// TwinCAT 3 PLC project PLC1
// ProgramVersion: 3.1.4023.0
// libraries:
//   Tc2_Standard, * (Beckhoff Automation GmbH)
//   Tc2_System, * (Beckhoff Automation GmbH)
//   Tc2_Utilities, * (Beckhoff Automation GmbH)
//   Tc3_Database, * (Beckhoff Automation GmbH)
//   Tc3_EventLogger, * (Beckhoff Automation GmbH)
//   Tc3_Module, * (Beckhoff Automation GmbH)
// project tree:
//   DUTs/ aE_Mode.TcDUT, aE_ProcessState.TcDUT, aE_State.TcDUT, aS_AnalogAlarm.TcDUT, aS_AutoControl.TcDUT, aS_DBField.TcDUT, aT_Furnace.TcDUT, aT_Heater.TcDUT, aT_Tank.TcDUT, aT_Turbine.TcDUT, AutoCtrlCmds.TcDUT, Components.TcDUT, InStream.TcDUT, MainInterface.TcDUT, OutStream.TcDUT, aS_PidParameter.TcDUT, Parameters.TcDUT
//   GVLs/ AlarmLimit.TcGVL, Interfacex.TcGVL, Streams.TcGVL
//   / PlcDBTask.TcTTO, PlcTask.TcTTO
//   POUs/ AlarmManagement.TcPOU, AutoControl.TcPOU, PnID.TcPOU, SaveDatabase.TcPOU, TanksSimulation.TcPOU, UpdateInterface.TcPOU
//   POUs/FB/ aFb_Motor.TcPOU, aFB_Valve.TcPOU
// real-time tasks:
//   TASK PlcTask: cycle T#100000us, priority 20, ADS port 350
//   TASK PlcDBTask: cycle T#1ms, priority 21, ADS port 351
//   TASK PlcTask1: cycle T#1ms, priority 22, ADS port 352
// I/O:
//   DEVICE Device 1 (EtherCAT), AmsNetId 5.57.208.6.2.1
//     Term 1 (EK1200) [EK1200-5000 EtherCAT Power supply (2A E-Bus)]
//       Term 2 (EL1004) [EL1004 4Ch. Dig. Input 24V, 3ms]
//       Term 3 (EL2004) [EL2004 4Ch. Dig. Output 24V, 0.5A]
//       Term 8 (EL3054) [EL3054 4Ch. Ana. Input 4-20mA]
//       Term 4 (EL9011) [EL9011 End Terminal]
//   DEVICE Device 5 (COM Port) (disabled)
// variable links:
//   PLC1/PLC1 Instance <-> Device 1 (EtherCAT)/Term 1 (EK1200)/Term 2 (EL1004)
//     PlcTask Inputs/AutoControl.bEmerNC <-> Channel 4/Input
//     PlcTask Inputs/AutoControl.bStart <-> Channel 3/Input
//     PlcTask Inputs/PnID.bHI <-> Channel 2/Input
//     PlcTask Inputs/PnID.bLO <-> Channel 1/Input
//   PLC1/PLC1 Instance <-> Device 1 (EtherCAT)/Term 1 (EK1200)/Term 3 (EL2004)
//     PlcTask Outputs/AutoControl.bErr <-> Channel 4/Output
//     PlcTask Outputs/AutoControl.bRun <-> Channel 3/Output
//     PlcTask Outputs/PnID.bMotor1 <-> Channel 1/Output
//     PlcTask Outputs/PnID.bMotor2 <-> Channel 2/Output
//   PLC1/PLC1 Instance <-> Device 1 (EtherCAT)/Term 1 (EK1200)/Term 8 (EL3054)
//     PlcTask Inputs/PnID.CircularPumpFlow <-> AI Standard Channel 1/Value

CONFIGURATION PLC1
    RESOURCE PLC ON TwinCAT3
        TASK PlcDBTask(INTERVAL := T#1ms, PRIORITY := 21);
        TASK PlcTask(INTERVAL := T#100000us, PRIORITY := 20);
        PROGRAM SaveDatabase WITH PlcDBTask : SaveDatabase;
        PROGRAM AutoControl WITH PlcTask : AutoControl;
        PROGRAM PnID WITH PlcTask : PnID;
        PROGRAM AlarmManagement WITH PlcTask : AlarmManagement;
        PROGRAM UpdateInterface WITH PlcTask : UpdateInterface;
    END_RESOURCE
END_CONFIGURATION

// ---- DUTs/aE_Mode.TcDUT
{attribute 'qualified_only'}
{attribute 'strict'}
TYPE aE_Mode :
(
	Manual := 1,
	Auto := 2,
	Service := 3
);
END_TYPE

// ---- DUTs/aE_ProcessState.TcDUT
{attribute 'qualified_only'}
{attribute 'strict'}
TYPE aE_ProcessState :
(
	Error := 0,
	Init := 1,
	Enable := 2,
	Start := 3,
	SteadyState := 4,
	Stop := 5,
	Disable := 6,
	Reset := 7
);
END_TYPE

// ---- DUTs/aE_State.TcDUT
{attribute 'qualified_only'}
{attribute 'strict'}
TYPE aE_State :
(
	Fault := 0,
	Auto := 1,
	ManRun := 2,
	ManStop := 3
);
END_TYPE

// ---- DUTs/aS_AnalogAlarm.TcDUT
TYPE aS_AnalogAlarm :
STRUCT
	HIHI: REAL;
	HI: REAL;
	LO: REAL;
	LOLO: REAL;
	Deadband: REAL;
END_STRUCT
END_TYPE

// ---- DUTs/aS_AutoControl.TcDUT
TYPE aS_AutoControl :
STRUCT
	Start: BOOL;
	Stop: BOOL;
	Setpoint: LREAL;
	ControlSignal: LREAL;
	Switch: BYTE;
END_STRUCT
END_TYPE

// ---- DUTs/aS_DBField.TcDUT
TYPE aS_DBField :
STRUCT
	Id: LINT;
	Sync: BOOL;
	Timestamp: DT;
	FurTemp: REAL;
	FurInper: REAL;
	LphTemp: REAL;
	LphPress: REAL;
	LphInpress: REAL;
	LphInflow: REAL;
	DeaTemp: REAL;
	DeaPress: REAL;
	HphTemp: REAL;
	HphPress: REAL;
	HphInpress: REAL;
	HphInflow: REAL;
	BoiTemp: REAL;
	BoiPress: REAL;
	ConTemp: REAL;
	ConInflow: REAL;
	TurHtemp: REAL;
	TurItemp: REAL;
	TurLtemp: REAL;
	TurHpress: REAL;
	TurIpress: REAL;
	TurLpress: REAL;
	TurSpeed: REAL;
	
	PconMode: BYTE;
	PconRun: BOOL;
	PconVal: REAL;
	PconTime: DINT;
	PconAtime: DINT;
	PconFault: BOOL;
	
	PsupMode: BYTE;
	PsupRun: BOOL;
	PsupVal: REAL;
	PsupTime: DINT;
	PsupAtime: DINT;
	PsupFault: BOOL;
	
	PcirMode: BYTE;
	PcirRun: BOOL;
	PcirVal: REAL;
	PcirTime: DINT;
	PcirAtime: DINT;
	PcirFault: BOOL;
	
	F1Mode: BYTE;
	F1Run: BOOL;
	F1Val: REAL;
	F1Time: DINT;
	F1Atime: DINT;
	F1Fault: BOOL;
	
	F2Mode: BYTE;
	F2Run: BOOL;
	F2Val: REAL;
	F2Time: DINT;
	F2Atime: DINT;
	F2Fault: BOOL;
	
	F3Mode: BYTE;
	F3Run: BOOL;
	F3Val: REAL;
	F3Time: DINT;
	F3Atime: DINT;
	F3Fault: BOOL;
	
	VlphMode: BYTE;
	VlphRun: BOOL;
	VlphVal: REAL;
	VlphTime: DINT;
	VlphAtime: DINT;
	VlphFault: BOOL;
	
	VdeaMode: BYTE;
	VdeaRun: BOOL;
	VdeaVal: REAL;
	VdeaTime: DINT;
	VdeaAtime: DINT;
	VdeaFault: BOOL;
	
	VhphMode: BYTE;
	VhphRun: BOOL;
	VhphVal: REAL;
	VhphTime: DINT;
	VhphAtime: DINT;
	VhphFault: BOOL;
	
	VturMode: BYTE;
	VturRun: BOOL;
	VturVal: REAL;
	VturTime: DINT;
	VturAtime: DINT;
	VturFault: BOOL;
	
	PintMode: BYTE;
	PintRun: BOOL;
	PintVal: REAL;
	PintTime: DINT;
	PintAtime: DINT;
	PintFault: BOOL;
END_STRUCT
END_TYPE

// ---- DUTs/aT_Furnace.TcDUT
TYPE aT_Furnace :
STRUCT
	InPercent: REAL;
	Temperature: REAL;
END_STRUCT
END_TYPE

// ---- DUTs/aT_Heater.TcDUT
TYPE aT_Heater :
STRUCT
	InPressure: REAL;
	InFlow: REAL;
	Temperature: REAL;
	Pressure: REAL;
END_STRUCT
END_TYPE

// ---- DUTs/aT_Tank.TcDUT
TYPE aT_Tank :
STRUCT
	HI: BOOL;
	LO: BOOL;
	Level: REAL;
END_STRUCT
END_TYPE

// ---- DUTs/aT_Turbine.TcDUT
TYPE aT_Turbine :
STRUCT
	Rotation: REAL;
	HighPressure: REAL;
	ImmediatePressure: REAL;
	OutPressure: REAL;
	HighTemperature: REAL;
	ImmediateTemperature: REAL;
	OutTemperature: REAL;
END_STRUCT
END_TYPE

// ---- DUTs/AutoCtrlCmds.TcDUT
TYPE AutoCtrlCmds :
STRUCT
	Start: BOOL;
	Stop: BOOL;
	Emergency: BOOL;
	Reset: BOOL;
	
	ProcessReady: BOOL;
	ProcessRun: BOOL;
	ProcessFault: BOOL;
END_STRUCT
END_TYPE

// ---- DUTs/Components.TcDUT
TYPE Components :
STRUCT
	ForceFan1: aFb_Motor;
	ForceFan2: aFb_Motor;
	ForceFan3: aFb_Motor;
	
	CondensePump: aFb_Motor;
	SupplyPump: aFb_Motor;
	CircularPump: aFb_Motor;
	InterPump: aFb_Motor;

	LPHValve: aFb_Valve;
	AirEjValve: aFb_Valve;
	HPHValve: aFb_Valve;
	TurbineValve: aFb_Valve;
	
	Furnace: aT_Furnace;
	LPHeater: aT_Heater;
	Deaerator: aT_Heater;
	HPHeater: aT_Heater;
	Boiler: aT_Heater;
	Turbine: aT_Turbine;
	Condenser: aT_Heater;
	
	InterTank: aT_Tank;
END_STRUCT
END_TYPE

// ---- DUTs/InStream.TcDUT
TYPE InStream :
STRUCT
	ForceFan1_Speed: REAL;
	ForceFan2_Speed: REAL;
	ForceFan3_Speed: REAL;
	Furnace_Temp: REAL;
	CondensePump_Press: REAL;
	CondensePump_Flow: REAL;
	CondensePump_Speed: REAL;
	LPHeater_Temp: REAL;
	LPHeater_Press: REAL;
	AirEjector_Temp: REAL;
	AirEjector_Press: REAL;
	SupplyPump_Press: REAL;
	SupplyPump_Flow: REAL;
	SupplyPump_Speed: REAL;
	HPHeater_Temp: REAL;
	HPHeater_Press: REAL;
	Boiler_Temp: REAL;
	Boiler_Press: REAL;
	Turbine_Rotation: REAL;
	Turbine_HighPress: REAL;
	Turbine_ImmediatePress: REAL;
	Turbine_OutPress: REAL;
	Turbine_HighTemp: REAL;
	Turbine_ImmediateTemp: REAL;
	Turbine_OutTemp: REAL;
	Condenser_Temp: REAL;

END_STRUCT
END_TYPE

// ---- DUTs/MainInterface.TcDUT
TYPE MainInterface :
STRUCT
	Components: Components;
END_STRUCT
END_TYPE

// ---- DUTs/OutStream.TcDUT
TYPE OutStream :
STRUCT
	ForceFan1_SetSpeed: REAL;
	ForceFan2_SetSpeed: REAL;
	ForceFan3_SetSpeed: REAL;
	CondensePump_SetSpeed: REAL;
	SupplyPump_SetSpeed: REAL;
	CircularPump_OutFlow: REAL;
	LPHeaterValve_SetPercent: REAL;
	AirEjectorValve_SetPercent: REAL;
	HPHeaterValve_SetPercent: REAL;
	TurbineValve_SetPercent: REAL;
END_STRUCT
END_TYPE

// ---- DUTs/aS_PidParameter.TcDUT
TYPE aS_PidParameter :
STRUCT
	Kp: LREAL;
	Ti: LREAL;
	Td: LREAL;
	Tn: LREAL;
END_STRUCT
END_TYPE

// ---- DUTs/Parameters.TcDUT
TYPE Parameters :
STRUCT
	PID_CondensePump_Press: aS_PidParameter := (Kp:= 91.7, Ti:= 6.368, Td:= 0.1396, Tn:= 0.078);//(Kp:= 91.7, Ti:= 6.368, Td:= 0.1396, Tn:= 0.078);//(Kp:= 200, Ti:= 33.333, Td:= 0, Tn:= 0.05);
	PID_SupplyPump_Press: aS_PidParameter := (Kp:= 40, Ti:= 10, Td:= 0.05, Tn:= 0.05);//(Kp:= 40, Ti:= 8, Td:= 0.125, Tn:= 0.05);
	//PID_Condenser_Temp: aS_PidParameter := (Kp:= -40, Ti:= 53.333, Td:= 2.5, Tn:= 0.05);
	PID_LPHeater_Temp: aS_PidParameter := (Kp:= 0.015, Ti:= 3, Td:= 0, Tn:= 0.05);//(Kp:= 0.02, Ti:= 6.667, Td:= 2, Tn:= 0.5);
	PID_AirEjector_Temp: aS_PidParameter := (Kp:= 0.025, Ti:= 50, Td:= 0, Tn:= 0.05);//(Kp:= 0.0085, Ti:= 4.048, Td:= 0, Tn:= 0.5);
	PID_HPHeater_Temp: aS_PidParameter := (Kp:= 0.01, Ti:= 20, Td:= 0, Tn:= 0.05);//(Kp:= 0.0103, Ti:= 4.12, Td:= 0, Tn:= 0.5);
	PID_Turbine_Speed: aS_PidParameter := (Kp:= 0.003, Ti:= 30, Td:= 0, Tn:= 0.05);//(Kp:= 0.001, Ti:= 10, Td:= 100, Tn:= 100);
	PID_Boiler_Temp: aS_PidParameter := (Kp:= 8, Ti:= 100, Td:= 0.0625, Tn:= 0.05);//(Kp:= 7, Ti:= 20, Td:= 1.4286, Tn:= 0.05);// //(Kp:= 7, Ti:= 100, Td:= 0, Tn:= 0.05);
	
	MaxSpeed_CondensePump: REAL := 1485;
	MaxSpeed_SupplyPump: REAL := 5645;
	MaxSpeed_CircularPump: REAL := 1500;
	MaxSpeed_InterPump: REAL := 1500;	
	MaxSpeed_ForceFan1: REAL := 1485;
	MaxSpeed_ForceFan2: REAL := 1485;
	MaxSpeed_ForceFan3: REAL := 1485;
	
	Condenser_Htemp: REAL := 50;
	Condenser_Ltemp: REAL := 30;
	
	SampleTime: REAL := 0.1;
END_STRUCT
END_TYPE

// ---- GVLs/AlarmLimit.TcGVL
{attribute 'qualified_only'}
VAR_GLOBAL
	alLPHeaterTemp: aS_AnalogAlarm := (HIHI:= 160, HI:= 150, LO:= 130, LOLO:= 120, Deadband:= 5);
	alLPHeaterPress: aS_AnalogAlarm := (HIHI:= 34, HI:= 31, LO:= 25, LOLO:= 22, Deadband:= 1);
	alDeaeratorTemp: aS_AnalogAlarm := (HIHI:= 220, HI:= 210, LO:= 190, LOLO:= 180, Deadband:= 5);
	alHPHeaterTemp: aS_AnalogAlarm := (HIHI:= 315, HI:= 305, LO:= 285, LOLO:= 275, Deadband:= 5);
	alHPHeaterPress: aS_AnalogAlarm := (HIHI:= 315, HI:= 305, LO:= 285, LOLO:= 275, Deadband:= 5);
	alBoilerTemp: aS_AnalogAlarm := (HIHI:= 590, HI:= 580, LO:= 550, LOLO:= 540, Deadband:= 5);
	alCondenserTemp: aS_AnalogAlarm := (HIHI:= 80, HI:= 70, LO:= 10, LOLO:= 5, Deadband:= 5);
	alTurbineTemp: aS_AnalogAlarm := (HIHI:= 170, HI:= 160, LO:= 140, LOLO:= 130, Deadband:= 5);
	alTurbinePress: aS_AnalogAlarm := (HIHI:= 0.2, HI:= 0.1, LO:= 0.02, LOLO:= 0.01, Deadband:= 0.005);
	alTurbineRotation: aS_AnalogAlarm := (HIHI:= 3020, HI:= 3010, LO:= 2990, LOLO:= 2980, Deadband:= 5);

END_VAR

// ---- GVLs/Interfacex.TcGVL
{attribute 'qualified_only'}
VAR_GLOBAL
	ScadaInterface: MainInterface;
	AutoCtrlCmds: AutoCtrlCmds;
	Parameters: Parameters;
END_VAR

// ---- GVLs/Streams.TcGVL
{attribute 'qualified_only'}
VAR_GLOBAL
	OutStream AT %MD0: OutStream;
	InStream AT %MD10: InStream;
END_VAR

// ---- POUs/SaveDatabase.TcPOU
PROGRAM SaveDatabase
VAR
	fbPLCDBWrite : FB_PLCDBWriteEvt (sNetID := '', tTimeout := T#5S);
	myDBID : UDINT:=1;
	sMyTableName : T_MaxString:='Data';
	ColumnNames : ARRAY [0..91] OF STRING(50);
	insertData : aS_DBField;
	tcMessage : I_TcMessage;
	
	//Các biến tạo timestamp
	systime: GETSYSTEMTIME;
	currentTime: T_FILETIME;
	timestring: string;
	
	bFirstScan: BOOL;
	bExecute: BOOL;
	fbTon: TON;
	iID: LINT;
END_VAR

IF NOT bFirstScan THEN
	bFirstScan := TRUE;
	InitColumnNames();
END_IF

fbTon(IN:= NOT fbTon.Q, PT:= T#1S);	
IF fbTon.Q THEN
	UpdateData();
	bExecute := TRUE;
END_IF

IF bExecute AND bFirstScan THEN
	//UpdateData();
	IF fbPLCDBWrite.WriteStruct(
		hDBID:= myDBID,
		sTableName:= sMyTableName,
		pRecord:= ADR(insertData),
		cbRecord:= SIZEOF(insertData),
		pColumnNames:= ADR(ColumnNames) ,
		cbColumnNames:= SIZEOF(ColumnNames)
	)
	THEN
		IF fbPLCDBWrite.bError THEN
			tcMessage := fbPLCDBWrite.ipTcResult;
		ELSE
			iId := iId + 1;
			bExecute:= FALSE;
		END_IF
	END_IF	
	
END_IF

ACTION InitColumnNames:
ColumnNames[0] := 'Id';
ColumnNames[1] := 'Sync';
ColumnNames[2] := 'Timestamp';

ColumnNames[3] := 'FurTemp';
ColumnNames[4] := 'FurInper';
ColumnNames[5] := 'LphTemp';
ColumnNames[6] := 'LphPress';
ColumnNames[7] := 'LphInpress';
ColumnNames[8] := 'LphInflow';
ColumnNames[9] := 'DeaTemp';
ColumnNames[10] := 'DeaPress';
ColumnNames[11] := 'HphTemp';
ColumnNames[12] := 'HphPress';
ColumnNames[13] := 'HphInpress';
ColumnNames[14] := 'HphInflow';
ColumnNames[15] := 'BoiTemp';
ColumnNames[16] := 'BoiPress';
ColumnNames[17] := 'ConTemp';
ColumnNames[18] := 'ConInflow';
ColumnNames[19] := 'TurHtemp';
ColumnNames[20] := 'TurItemp';
ColumnNames[21] := 'TurLtemp';
ColumnNames[22] := 'TurHpress';
ColumnNames[23] := 'TurIpress';
ColumnNames[24] := 'TurLpress';
ColumnNames[25] := 'TurSpeed';

ColumnNames[26] := 'PconMode';
ColumnNames[27] := 'PconRun';
ColumnNames[28] := 'PconVal';
ColumnNames[29] := 'PconTime';
ColumnNames[30] := 'PconAtime';
ColumnNames[31] := 'PconFault';

ColumnNames[32] := 'PsupMode';
ColumnNames[33] := 'PsupRun';
ColumnNames[34] := 'PsupVal';
ColumnNames[35] := 'PsupTime';
ColumnNames[36] := 'PsupAtime';
ColumnNames[37] := 'PsupFault';

ColumnNames[38] := 'PcirMode';
ColumnNames[39] := 'PcirRun';
ColumnNames[40] := 'PcirVal';
ColumnNames[41] := 'PcirTime';
ColumnNames[42] := 'PcirAtime';
ColumnNames[43] := 'PcirFault';

ColumnNames[44] := 'F1Mode';
ColumnNames[45] := 'F1Run';
ColumnNames[46] := 'F1Val';
ColumnNames[47] := 'F1Time';
ColumnNames[48] := 'F1Atime';
ColumnNames[49] := 'F1Fault';

ColumnNames[50] := 'F2Mode';
ColumnNames[51] := 'F2Run';
ColumnNames[52] := 'F2Val';
ColumnNames[53] := 'F2Time';
ColumnNames[54] := 'F2Atime';
ColumnNames[55] := 'F2Fault';

ColumnNames[56] := 'F3Mode';
ColumnNames[57] := 'F3Run';
ColumnNames[58] := 'F3Val';
ColumnNames[59] := 'F3Time';
ColumnNames[60] := 'F3Atime';
ColumnNames[61] := 'F3Fault';

ColumnNames[62] := 'VlphMode';
ColumnNames[63] := 'VlphRun';
ColumnNames[64] := 'VlphVal';
ColumnNames[65] := 'VlphTime';
ColumnNames[66] := 'VlphAtime';
ColumnNames[67] := 'VlphFault';

ColumnNames[68] := 'VdeaMode';
ColumnNames[69] := 'VdeaRun';
ColumnNames[70] := 'VdeaVal';
ColumnNames[71] := 'VdeaTime';
ColumnNames[72] := 'VdeaAtime';
ColumnNames[73] := 'VdeaFault';

ColumnNames[74] := 'VhphMode';
ColumnNames[75] := 'VhphRun';
ColumnNames[76] := 'VhphVal';
ColumnNames[77] := 'VhphTime';
ColumnNames[78] := 'VhphAtime';
ColumnNames[79] := 'VhphFault';

ColumnNames[80] := 'VturMode';
ColumnNames[81] := 'VturRun';
ColumnNames[82] := 'VturVal';
ColumnNames[83] := 'VturTime';
ColumnNames[84] := 'VturAtime';
ColumnNames[85] := 'VturFault';

ColumnNames[86] := 'PintMode';
ColumnNames[87] := 'PintRun';
ColumnNames[88] := 'PintVal';
ColumnNames[89] := 'PintTime';
ColumnNames[90] := 'PintAtime';
ColumnNames[91] := 'PintFault';
END_ACTION

ACTION UpdateData:
systime(timeLoDW => currentTime.dwLowDateTime, timeHiDW => currentTime.dwHighDateTime);	
timestring:= DT_TO_STRING(FILETIME_TO_DT(currentTime));
timestring:= delete(timestring, 3, 1);
timestring:= replace(timestring, ' ', 1, 11);

insertData.Id := iID;
insertData.Sync := FALSE;
insertData.Timestamp:= FILETIME_TO_DT(currentTime);
insertData.FurTemp:= Interfacex.ScadaInterface.Components.Furnace.Temperature;
insertData.FurInper:= Interfacex.ScadaInterface.Components.Furnace.InPercent;
insertData.LphTemp:= Interfacex.ScadaInterface.Components.LPHeater.Temperature;
insertData.LphPress:= Interfacex.ScadaInterface.Components.LPHeater.Pressure;
insertData.LphInpress:= Interfacex.ScadaInterface.Components.LPHeater.InPressure;
insertData.LphInflow:= Interfacex.ScadaInterface.Components.LPHeater.InFlow;
insertData.DeaTemp:= Interfacex.ScadaInterface.Components.Deaerator.Temperature;
insertData.DeaPress:= Interfacex.ScadaInterface.Components.Deaerator.Pressure;
insertData.HphTemp:= Interfacex.ScadaInterface.Components.HPHeater.Temperature;
insertData.HphPress:= Interfacex.ScadaInterface.Components.HPHeater.Pressure;
insertData.HphInpress:= Interfacex.ScadaInterface.Components.HPHeater.InPressure;
insertData.HphInflow:= Interfacex.ScadaInterface.Components.HPHeater.InFlow;
insertData.BoiTemp:= Interfacex.ScadaInterface.Components.Boiler.Temperature;
insertData.BoiPress:= Interfacex.ScadaInterface.Components.Boiler.Pressure;
insertData.ConTemp:= Interfacex.ScadaInterface.Components.Condenser.Temperature;
insertData.ConInflow:= Interfacex.ScadaInterface.Components.Condenser.InFlow;
insertData.TurHtemp:= Interfacex.ScadaInterface.Components.Turbine.HighTemperature;
insertData.TurItemp:= Interfacex.ScadaInterface.Components.Turbine.ImmediateTemperature;
insertData.TurLtemp:= Interfacex.ScadaInterface.Components.Turbine.OutTemperature;
insertData.TurHpress:= Interfacex.ScadaInterface.Components.Turbine.HighPressure;
insertData.TurIpress:= Interfacex.ScadaInterface.Components.Turbine.ImmediatePressure;
insertData.TurLpress:= Interfacex.ScadaInterface.Components.Turbine.OutPressure;
insertData.TurSpeed:= Interfacex.ScadaInterface.Components.Turbine.Rotation;

insertData.PconMode:= INT_TO_BYTE(Interfacex.ScadaInterface.Components.CondensePump.Mode); 
insertData.PconRun:= Interfacex.ScadaInterface.Components.CondensePump.RunFeedback;
insertData.PconVal:= Interfacex.ScadaInterface.Components.CondensePump.ActualSpeed;
insertData.PconTime:= Interfacex.ScadaInterface.Components.CondensePump.Runtime;
insertData.PconAtime:= Interfacex.ScadaInterface.Components.CondensePump.AccRuntime;
insertData.PconFault:= Interfacex.ScadaInterface.Components.CondensePump.Fault;

insertData.PsupMode:= INT_TO_BYTE(Interfacex.ScadaInterface.Components.SupplyPump.Mode); 
insertData.PsupRun:= Interfacex.ScadaInterface.Components.SupplyPump.RunFeedback;
insertData.PsupVal:= Interfacex.ScadaInterface.Components.SupplyPump.ActualSpeed;
insertData.PsupTime:= Interfacex.ScadaInterface.Components.SupplyPump.Runtime;
insertData.PsupAtime:= Interfacex.ScadaInterface.Components.SupplyPump.AccRuntime;
insertData.PsupFault:= Interfacex.ScadaInterface.Components.SupplyPump.Fault;

insertData.PcirMode:= INT_TO_BYTE(Interfacex.ScadaInterface.Components.CircularPump.Mode); 
insertData.PcirRun:= Interfacex.ScadaInterface.Components.CircularPump.RunFeedback;
insertData.PcirVal:= Interfacex.ScadaInterface.Components.CircularPump.ActualSpeed;
insertData.PcirTime:= Interfacex.ScadaInterface.Components.CircularPump.Runtime;
insertData.PcirAtime:= Interfacex.ScadaInterface.Components.CircularPump.AccRuntime;
insertData.PcirFault:= Interfacex.ScadaInterface.Components.CircularPump.Fault;

insertData.F1Mode:= INT_TO_BYTE(Interfacex.ScadaInterface.Components.ForceFan1.Mode); 
insertData.F1Run:= Interfacex.ScadaInterface.Components.ForceFan1.RunFeedback;
insertData.F1Val:= Interfacex.ScadaInterface.Components.ForceFan1.ActualSpeed;
insertData.F1Time:= Interfacex.ScadaInterface.Components.ForceFan1.Runtime;
insertData.F1Atime:= Interfacex.ScadaInterface.Components.ForceFan1.AccRuntime;
insertData.F1Fault:= Interfacex.ScadaInterface.Components.ForceFan1.Fault;

insertData.F2Mode:= INT_TO_BYTE(Interfacex.ScadaInterface.Components.ForceFan2.Mode); 
insertData.F2Run:= Interfacex.ScadaInterface.Components.ForceFan2.RunFeedback;
insertData.F2Val:= Interfacex.ScadaInterface.Components.ForceFan2.ActualSpeed;
insertData.F2Time:= Interfacex.ScadaInterface.Components.ForceFan2.Runtime;
insertData.F2Atime:= Interfacex.ScadaInterface.Components.ForceFan2.AccRuntime;
insertData.F2Fault:= Interfacex.ScadaInterface.Components.ForceFan2.Fault;

insertData.F3Mode:= INT_TO_BYTE(Interfacex.ScadaInterface.Components.ForceFan3.Mode); 
insertData.F3Run:= Interfacex.ScadaInterface.Components.ForceFan3.RunFeedback;
insertData.F3Val:= Interfacex.ScadaInterface.Components.ForceFan3.ActualSpeed;
insertData.F3Time:= Interfacex.ScadaInterface.Components.ForceFan3.Runtime;
insertData.F3Atime:= Interfacex.ScadaInterface.Components.ForceFan3.AccRuntime;
insertData.F3Fault:= Interfacex.ScadaInterface.Components.ForceFan3.Fault;

insertData.VlphMode:= INT_TO_BYTE(Interfacex.ScadaInterface.Components.LPHValve.Mode); 
insertData.VlphRun:= Interfacex.ScadaInterface.Components.LPHValve.RunFeedback;
insertData.VlphVal:= Interfacex.ScadaInterface.Components.LPHValve.OpenPercent;
insertData.VlphTime:= Interfacex.ScadaInterface.Components.LPHValve.Runtime;
insertData.VlphAtime:= Interfacex.ScadaInterface.Components.LPHValve.AccRuntime;
insertData.VlphFault:= Interfacex.ScadaInterface.Components.LPHValve.Fault;

insertData.VdeaMode:= INT_TO_BYTE(Interfacex.ScadaInterface.Components.AirEjValve.Mode); 
insertData.VdeaRun:= Interfacex.ScadaInterface.Components.AirEjValve.RunFeedback;
insertData.VdeaVal:= Interfacex.ScadaInterface.Components.AirEjValve.OpenPercent;
insertData.VdeaTime:= Interfacex.ScadaInterface.Components.AirEjValve.Runtime;
insertData.VdeaAtime:= Interfacex.ScadaInterface.Components.AirEjValve.AccRuntime;
insertData.VdeaFault:= Interfacex.ScadaInterface.Components.AirEjValve.Fault;

insertData.VhphMode:= INT_TO_BYTE(Interfacex.ScadaInterface.Components.HPHValve.Mode); 
insertData.VhphRun:= Interfacex.ScadaInterface.Components.HPHValve.RunFeedback;
insertData.VhphVal:= Interfacex.ScadaInterface.Components.HPHValve.OpenPercent;
insertData.VhphTime:= Interfacex.ScadaInterface.Components.HPHValve.Runtime;
insertData.VhphAtime:= Interfacex.ScadaInterface.Components.HPHValve.AccRuntime;
insertData.VhphFault:= Interfacex.ScadaInterface.Components.HPHValve.Fault;

insertData.VturMode:= INT_TO_BYTE(Interfacex.ScadaInterface.Components.TurbineValve.Mode); 
insertData.VturRun:= Interfacex.ScadaInterface.Components.TurbineValve.RunFeedback;
insertData.VturVal:= Interfacex.ScadaInterface.Components.TurbineValve.OpenPercent;
insertData.VturTime:= Interfacex.ScadaInterface.Components.TurbineValve.Runtime;
insertData.VturAtime:= Interfacex.ScadaInterface.Components.TurbineValve.AccRuntime;
insertData.VturFault:= Interfacex.ScadaInterface.Components.TurbineValve.Fault;

insertData.PintMode:= INT_TO_BYTE(Interfacex.ScadaInterface.Components.InterPump.Mode); 
insertData.PintRun:= Interfacex.ScadaInterface.Components.InterPump.RunFeedback;
insertData.PintVal:= Interfacex.ScadaInterface.Components.InterPump.ActualSpeed;
insertData.PintTime:= Interfacex.ScadaInterface.Components.InterPump.Runtime;
insertData.PintAtime:= Interfacex.ScadaInterface.Components.InterPump.AccRuntime;
insertData.PintFault:= Interfacex.ScadaInterface.Components.InterPump.Fault;
END_ACTION

END_PROGRAM

// ---- POUs/AutoControl.TcPOU
PROGRAM AutoControl
VAR_INPUT
	bStart AT %I* : BOOL;
	bEmerNC AT %I*: BOOL := TRUE;
END_VAR	
VAR_OUTPUT
	bRun AT %Q*: BOOL;
	bErr AT %Q*: BOOL;
END_VAR
VAR
	{region 'Control Template'} 			//Struct to manipulate the auto mode 
	CondensePump_Press: aS_AutoControl;
	SupplyPump_Press: aS_AutoControl;
	Condenser_Temp: aS_AutoControl;
	LPHeater_Temp: aS_AutoControl;
	AirEjector_Temp: aS_AutoControl;
	HPHeater_Temp: aS_AutoControl;
	Turbine_Speed: aS_AutoControl;
	Boiler_Temp: aS_AutoControl;
	InterTank_Level: aS_AutoControl;
	{endregion}
		 
	{region 'Component PID Controllers'}
	ForceFan1_PID: FB_BasicPID;
	ForceFan2_PID: FB_BasicPID;
	ForceFan3_PID: FB_BasicPID;
	CondensePump_Press_PID: FB_BasicPID;
	SupplyPump_Press_PID: FB_BasicPID;
	//Condenser_Temp_PID: FB_BasicPID;
	LPHeater_Temp_PID: FB_BasicPID;
	AirEjector_Temp_PID: FB_BasicPID;
	HPHeater_Temp_PID: FB_BasicPID;
	Turbine_Speed_PID: FB_BasicPID;
	Boiler_Temp_PID: FB_BasicPID;

	ForceFan1_Trig: R_TRIG;
	ForceFan2_Trig: R_TRIG;
	ForceFan3_Trig: R_TRIG;
	CondensePump_Press_Trig: R_TRIG;
	SupplyPump_Press_Trig: R_TRIG;
	//Condenser_Temp_Trig: R_TRIG;
	LPHeater_Temp_Trig: R_TRIG;
	AirEjector_Temp_Trig: R_TRIG;
	HPHeater_Temp_Trig: R_TRIG;
	Turbine_Speed_Trig: R_TRIG;
	Boiler_Temp_Trig: R_TRIG;	 
	
	setpoint: REAL := 0.266;
	setpoint2: REAL := 28;
	setpoint3: REAL := 167;
	setpoint4: REAL := 37.85; //200,12.5,0.3,0.05
	setpoint5: REAL := 141.3;
	setpoint6: REAL := 200;
	setpoint7: REAL := 295;
	setpoint8: REAL := 3000;
	setpoint9: REAL := 566;
	{endregion}
		 
	{region 'Process State Vars'}
	ProcessState: aE_ProcessState := aE_ProcessState.Init;
	StartState: BYTE;
		 
	flag1: BOOL;
	flag2: BOOL;
	flag3: BOOL;
		 
	fbTon: TON;
	fbTon2: TON;
	{endregion}
		 
	
	{region 'Control Commands'}
	ProcessStart: BOOL;
	ProcessStop: BOOL;
	ProcessEmergency: BOOL;
	ProcessReset: BOOL;
		 
	ProcessReady: BOOL;
	ProcessRun: BOOL;
	ProcessFault: BOOL;
	
	bStateOn: BOOL := FALSE;
	trigBtnOn: R_TRIG;
	rtrigStateOn: R_TRIG;
	ftrigStateOn: F_TRIG;
	{endregion}
	i: INT;
	fbttemp: TON;
END_VAR

//Chú ý lỗi ở việc reset bộ pid

{region 'Control signal'}
IF Interfacex.AutoCtrlCmds.Start THEN
	bStateOn:= TRUE;
END_IF
IF ProcessFault OR Interfacex.AutoCtrlCmds.Stop THEN
	bStateOn:= FALSE;
END_IF
trigBtnOn(CLK:= bStart);
IF trigBtnOn.Q THEN
	bStateOn := NOT bStateOn;
END_IF
rtrigStateOn(CLK:= bStateOn);
ftrigStateOn(CLK:= bStateOn);

ProcessStart := Interfacex.AutoCtrlCmds.Start OR rtrigStateOn.Q;
ProcessStop := Interfacex.AutoCtrlCmds.Stop OR ftrigStateOn.Q;
ProcessEmergency := Interfacex.AutoCtrlCmds.Emergency OR NOT bEmerNC;
ProcessReset := Interfacex.AutoCtrlCmds.Reset OR rtrigStateOn.Q;
	 
Interfacex.AutoCtrlCmds.ProcessReady := ProcessReady;
Interfacex.AutoCtrlCmds.ProcessRun := ProcessRun;
Interfacex.AutoCtrlCmds.ProcessFault := ProcessFault;
{endregion}

{region 'Tank Simulation Handling'}
IF ProcessRun THEN 
	IF NOT PnID.bHI THEN
		InterTank_Level.Start:= FALSE;
		InterTank_Level.Stop:= TRUE;
	END_IF
	IF PnID.bLO THEN
		InterTank_Level.Start:= TRUE;
		InterTank_Level.Stop:= FALSE;		
	END_IF
	
	IF Streams.InStream.Condenser_Temp < 30 THEN
		Condenser_Temp.Start:= FALSE;
		Condenser_Temp.Stop:= TRUE;
	END_IF
	IF Streams.InStream.Condenser_Temp > 50 THEN
		Condenser_Temp.Start:= TRUE;
		Condenser_Temp.Stop:= FALSE;
	END_IF
//ELSE
//	Condenser_Temp.Start:= FALSE;
//	Condenser_Temp.Stop:= TRUE;
//	InterTank_Level.Start:= FALSE;
//	InterTank_Level.Stop:= TRUE;		
END_IF

bRun := ProcessRun;
bErr := ProcessFault;
{endregion}


{region 'Main State Machine'}
CASE ProcessState OF
	aE_ProcessState.Init:
		//Light
		ProcessReady := TRUE;
		ProcessRun := FALSE;
		ProcessFault := FALSE;
		//Reset all components and all PID Controllers
		Reset_StopAllComponents();
		ResetAllPidControllers();

		//Reset all flags and timers
		flag1 := FALSE;
		flag2 := FALSE;
		flag3 := FALSE;
		StartState := 0;
		fbTon(IN := FALSE);
		//Check if all conditions is matched
		//Next state
		IF ProcessEmergency THEN
			ProcessState := aE_ProcessState.Error;
		END_IF
		IF ProcessStart THEN
			ProcessState := aE_ProcessState.Enable;
		END_IF
		
	aE_ProcessState.Enable:
		//Light
		ProcessReady := FALSE;
		ProcessRun := TRUE;
		ProcessFault := FALSE;

		//Start all components and unlock all Pid controllers
		StartAllComponents();
		UnlockAllPidControllers();
		
		//Next state
		IF ProcessEmergency THEN
			ProcessState := aE_ProcessState.Error;
		END_IF
//		fbttemp(IN:= TRUE, PT:=T#3S);
//		IF fbttemp.Q THEN
			ProcessState := aE_ProcessState.Start;
//			fbttemp(IN:= FALSE);
//		END_IF
		
	aE_ProcessState.Start:
//		fbttemp(IN:= TRUE, PT:=T#3S);												//comment this!
//		IF fbttemp.Q THEN
//			ProcessState := aE_ProcessState.SteadyState;
//			fbttemp(IN:= FALSE);
//		END_IF
			 
		//Light
		ProcessReady := FALSE;
		ProcessRun := TRUE;
		ProcessFault := FALSE;

		IF ProcessEmergency THEN
			ProcessState := aE_ProcessState.Error;
		END_IF
	{region 'aa'}
		CASE StartState OF 
			0:  //Start state 0: increase condense pump pressure to 5 bar, supply pump pressure to 30 bar
				//Assign setpoint
				CondensePump_Press.Setpoint := 5;		//5 bar, pid control
				SupplyPump_Press.Setpoint := 30;		//10 bar, pid control
				//Condenser_Temp.Setpoint := 37.85;		//37.85 oC, pid control
				LPHeater_Temp.Setpoint := 100;			//100% valve openpercent, switch = direct control
				AirEjector_Temp.Setpoint := 100;		//100% valve openpercent, switch = direct control
				HPHeater_Temp.Setpoint := 72;			//100% valve openpercent, switch = direct control
				Turbine_Speed.Setpoint := 100;			//100% valve openpercent, switch = direct control
				Boiler_Temp.Setpoint := 37.85;			//37.85 oC, pid control		
				
				//Switch controller
				LPHeater_Temp.Switch := 0;
				AirEjector_Temp.Switch := 0;
				HPHeater_Temp.Switch := 0;
				Turbine_Speed.Switch := 0;
				
				//Check condition to change state
				IF Streams.InStream.CondensePump_Press >= 5 THEN
					flag1 := TRUE;
				END_IF
				IF Streams.InStream.SupplyPump_Press >= 10 THEN
					flag2 := TRUE;
				END_IF
				IF flag1 = TRUE AND flag2 = TRUE THEN
					fbTon(IN := TRUE, PT:= T#5S);
					IF fbTon.Q THEN
						StartState := 1;
						flag1 := FALSE; flag2:= FALSE; 
						fbTon(IN := FALSE);
					END_IF
				END_IF
				
			1:  //Start state 1: increase boiler temp to 350 oC
				//Assign setpoint
				CondensePump_Press.Setpoint := 5;		//5 bar, pid control
				SupplyPump_Press.Setpoint := 30;		//10 bar, pid control
				//Condenser_Temp.Setpoint := 37.85;		//37.85 oC, pid control
				LPHeater_Temp.Setpoint := 100;			//100% valve openpercent, switch = direct control
				AirEjector_Temp.Setpoint := 100;		//100% valve openpercent, switch = direct control
				HPHeater_Temp.Setpoint := 72;			//100% valve openpercent, switch = direct control
				Turbine_Speed.Setpoint := 100;			//100% valve openpercent, switch = direct control
				Boiler_Temp.Setpoint := 350;			//37.85 oC, pid control		
				
				//Switch controller
				LPHeater_Temp.Switch := 0;
				AirEjector_Temp.Switch := 0;
				HPHeater_Temp.Switch := 0;
				Turbine_Speed.Switch := 0;
				
				//Check condition to change state
				IF Streams.InStream.Boiler_Temp >= 350 THEN
					flag1 := TRUE;
				END_IF
				IF flag1 = TRUE THEN
					fbTon(IN := TRUE, PT:= T#10S);
					IF fbTon.Q THEN
						StartState := 2;
						flag1 := FALSE; 
						fbTon(IN := FALSE);
					END_IF
				END_IF
				
			2:  //Start state 2: increase condense pump pressure to 15 bar, supply pump pressure to 100 bar
				//Assign setpoint
				CondensePump_Press.Setpoint := 15;		//15 bar, pid control
				SupplyPump_Press.Setpoint := 100;		//100 bar, pid control
				//Condenser_Temp.Setpoint := 37.85;		//37.85 oC, pid control
				LPHeater_Temp.Setpoint := 100;			//100% valve openpercent, switch = direct control
				AirEjector_Temp.Setpoint := 100;		//100% valve openpercent, switch = direct control
				HPHeater_Temp.Setpoint := 72;			//100% valve openpercent, switch = direct control
				Turbine_Speed.Setpoint := 100;			//100% valve openpercent, switch = direct control
				Boiler_Temp.Setpoint := 350;			//350 oC, pid control		
				
				//Switch controller
				LPHeater_Temp.Switch := 0;
				AirEjector_Temp.Switch := 0;
				HPHeater_Temp.Switch := 0;
				Turbine_Speed.Switch := 0;
				
				//Check condition to change state
				IF Streams.InStream.CondensePump_Press >= 15 THEN
					flag1 := TRUE;
				END_IF
				IF Streams.InStream.SupplyPump_Press >= 100 THEN
					flag2 := TRUE;
				END_IF
				IF flag1 = TRUE AND flag2 = TRUE THEN
					fbTon(IN := TRUE, PT:= T#5S);
					IF fbTon.Q THEN
						StartState := 3;
						flag1 := FALSE; flag2 := FALSE; 
						fbTon(IN := FALSE);
					END_IF
				END_IF		
				
			3:  //Start state 3: increase boiler temp to 450 oC
				//Assign setpoint
				CondensePump_Press.Setpoint := 15;		//5 bar, pid control
				SupplyPump_Press.Setpoint := 100;		//10 bar, pid control
				//Condenser_Temp.Setpoint := 37.85;		//37.85 oC, pid control
				LPHeater_Temp.Setpoint := 100;		//100% valve openpercent, switch = direct control
				AirEjector_Temp.Setpoint := 200;		//100% valve openpercent, switch = direct control
				HPHeater_Temp.Setpoint := 72;			//100% valve openpercent, switch = direct control
				Turbine_Speed.Setpoint := 100;			//100% valve openpercent, switch = direct control
				Boiler_Temp.Setpoint := 450;			//37.85 oC, pid control		
				
				//Switch controller
				LPHeater_Temp.Switch := 0;
				AirEjector_Temp.Switch := 1;
				HPHeater_Temp.Switch := 0;
				Turbine_Speed.Switch := 0;
				
				//Check condition to change state
				IF Streams.InStream.Boiler_Temp >= 450 THEN
					flag1 := TRUE;
				END_IF
				IF flag1 = TRUE THEN
					fbTon(IN := TRUE, PT:= T#10S);
					IF fbTon.Q THEN
						StartState := 4;
						flag1 := FALSE; 
						fbTon(IN := FALSE);
					END_IF
				END_IF
				
			4:  //Start state 4: increase condense pump pressure to 28 bar, supply pump pressure to 167 bar
				//Assign setpoint
				CondensePump_Press.Setpoint := 28;		//15 bar, pid control
				SupplyPump_Press.Setpoint := 167;		//100 bar, pid control
				//Condenser_Temp.Setpoint := 37.85;		//37.85 oC, pid control
				LPHeater_Temp.Setpoint := 100;			//100% valve openpercent, switch = direct control
				AirEjector_Temp.Setpoint := 200;		//100% valve openpercent, switch = direct control
				HPHeater_Temp.Setpoint := 72;			//100% valve openpercent, switch = direct control
				Turbine_Speed.Setpoint := 100;			//100% valve openpercent, switch = direct control
				Boiler_Temp.Setpoint := 450;			//350 oC, pid control		
				
				//Switch controller
				LPHeater_Temp.Switch := 0;
				AirEjector_Temp.Switch := 1;
				HPHeater_Temp.Switch := 0;
				Turbine_Speed.Switch := 0;
				
				//Check condition to change state
				IF Streams.InStream.CondensePump_Press >= 28 THEN
					flag1 := TRUE;
				END_IF
				IF Streams.InStream.SupplyPump_Press >= 167 THEN
					flag2 := TRUE;
				END_IF
				IF flag1 = TRUE AND flag2 = TRUE THEN
					fbTon(IN := TRUE, PT:= T#5S);
					IF fbTon.Q THEN
						StartState := 5;
						flag1 := FALSE; flag2 := FALSE;
						fbTon(IN := FALSE);
					END_IF
				END_IF	
			
			5:  //Start state 5: increase boiler temp to 566 oC
				//Assign setpoint
				CondensePump_Press.Setpoint := 28;		//15 bar, pid control
				SupplyPump_Press.Setpoint := 167;		//100 bar, pid control
				//Condenser_Temp.Setpoint := 37.85;		//37.85 oC, pid control
				LPHeater_Temp.Setpoint := 100;			//100% valve openpercent, switch = direct control
				AirEjector_Temp.Setpoint := 200;		//100% valve openpercent, switch = direct control
				HPHeater_Temp.Setpoint := 295;			//100% valve openpercent, switch = direct control
				Turbine_Speed.Setpoint := 100;			//100% valve openpercent, switch = direct control
				Boiler_Temp.Setpoint := 566;			//350 oC, pid control		
				
				//Switch controller
				LPHeater_Temp.Switch := 0;
				AirEjector_Temp.Switch := 1;
				HPHeater_Temp.Switch := 1;
				Turbine_Speed.Switch := 0;
				
				//Check condition to change state
				IF Streams.InStream.Boiler_Temp >= 550 THEN
					flag1 := TRUE;
				END_IF
				IF flag1 = TRUE THEN
					fbTon(IN := TRUE, PT:= T#5S);
					IF fbTon.Q THEN
						LPHeater_Temp.Setpoint := 141.3;			//100% valve openpercent, switch = direct control
						Turbine_Speed.Setpoint := 3000;			//100% valve openpercent, switch = direct control
						Turbine_Speed.Switch := 1;
						LPHeater_Temp.Switch := 1;
						fbTon2(IN := TRUE, PT:= T#90S);		//Steady State after 130s
						IF fbTon2.Q THEN
							StartState := 0;
							//Next state
							ProcessState := aE_ProcessState.SteadyState;
							flag1 := FALSE; 
							fbTon(IN := FALSE);
							fbTon2(IN:= FALSE);
						END_IF
					END_IF
				END_IF				
		END_CASE
		
		{endregion}
		  
		
	
	aE_ProcessState.SteadyState:
		//Light
		ProcessReady := FALSE;
		ProcessRun := TRUE;
		ProcessFault := FALSE;

		//Next State
		IF ProcessEmergency THEN
			ProcessState := aE_ProcessState.Error;
		END_IF
		IF ProcessStop THEN
			ProcessState := aE_ProcessState.Stop;
		END_IF
		
	aE_ProcessState.Stop:
		//Reset processstop
		//ProcessStop := FALSE;
		//Light
		ProcessReady := FALSE;
		ProcessRun := TRUE;
		ProcessFault := FALSE;
		
		//Stop process
		CondensePump_Press.Stop := TRUE;
		SupplyPump_Press.Stop := TRUE;
		//Condenser_Temp.Stop := TRUE;
		//InterTank_Level.Stop := TRUE;
		LPHeater_Temp.Stop := TRUE;
		AirEjector_Temp.Stop := TRUE;
		HPHeater_Temp.Stop := TRUE;
		Turbine_Speed.Stop := TRUE;
		Boiler_Temp.Stop := TRUE;

		//Next State
		IF ProcessEmergency THEN
			ProcessState := aE_ProcessState.Error;
		END_IF
//		fbttemp(IN:= TRUE, PT:=T#3S);
//		IF fbttemp.Q THEN
//			ProcessState := aE_ProcessState.Disable;
//			fbttemp(IN:= FALSE);
//		END_IF
		
		IF Streams.InStream.Boiler_Temp <= 45 THEN
			ProcessState := aE_ProcessState.Disable;
		END_IF
	aE_ProcessState.Disable:
		//Light
		ProcessReady := FALSE;
		ProcessRun := FALSE;
		ProcessFault := FALSE;

		//Stop all components and lock all Pid Controllers, Clear all start flags of components
		StopAllComponents();
		LockAllPidControllers();
		Reset_StartAllComponents();
		
		//Next State
		IF ProcessEmergency THEN
			ProcessState := aE_ProcessState.Error;
		END_IF
//		fbttemp(IN:= TRUE, PT:=T#3S);
//		IF fbttemp.Q THEN
			ProcessState := aE_ProcessState.Init;
//			fbttemp(IN:= FALSE);
//		END_IF
		
	aE_ProcessState.Error:
		//Light
		ProcessReady := FALSE;
		ProcessRun := FALSE;
		ProcessFault := TRUE;

	 	//Stop all components and clear start flags
		StopAllComponents();
		LockAllPidControllers();
		Reset_StartAllComponents();
		
		//Next State	 
		IF ProcessReset THEN
			ProcessState := aE_ProcessState.Reset;
		END_IF
		
	aE_ProcessState.Reset:
		//Light
		ProcessReady := FALSE;
		ProcessRun := FALSE;
		ProcessFault := TRUE;

		//Next State
		ProcessState := aE_ProcessState.Init;
END_CASE
{endregion}

{region 'Component Controllers'}
//IF (ProcessState = aE_ProcessState.Start OR ProcessState = aE_ProcessState.SteadyState OR ProcessState = aE_ProcessState.Stop) THEN 
	CondensePump_Press_PID(fSetpointValue := CondensePump_Press.Setpoint,
							fActualValue := Streams.InStream.CondensePump_Press,
							bReset := NOT PnID.CondensePump.Cmd OR CondensePump_Press.ResetPid,
							fCtrlCycleTime := Interfacex.Parameters.SampleTime,
							fKp := Interfacex.Parameters.PID_CondensePump_Press.Kp,
							fTn := Interfacex.Parameters.PID_CondensePump_Press.Ti,
							fTv := Interfacex.Parameters.PID_CondensePump_Press.Td,
							fTd := Interfacex.Parameters.PID_CondensePump_Press.Tn,
							fCtrlOutput => CondensePump_Press.ControlSignal);
								 
	SupplyPump_Press_PID(fSetpointValue := SupplyPump_Press.Setpoint,
							fActualValue := Streams.InStream.SupplyPump_Press,
							bReset := NOT PnID.SupplyPump.Cmd OR SupplyPump_Press.ResetPid,
							fCtrlCycleTime := Interfacex.Parameters.SampleTime,
							fKp := Interfacex.Parameters.PID_SupplyPump_Press.Kp,
							fTn := Interfacex.Parameters.PID_SupplyPump_Press.Ti,
							fTv := Interfacex.Parameters.PID_SupplyPump_Press.Td,
							fTd := Interfacex.Parameters.PID_SupplyPump_Press.Tn,
							fCtrlOutput => SupplyPump_Press.ControlSignal);	
		  
//	Condenser_Temp_PID(fSetpointValue := Condenser_Temp.Setpoint,
//							fActualValue := Streams.InStream.Condenser_Temp,
//							bReset := NOT PnID.CircularPump.Cmd OR Condenser_Temp.ResetPid,
//							fCtrlCycleTime := Interfacex.Parameters.SampleTime,
//							fKp := Interfacex.Parameters.PID_Condenser_Temp.Kp,
//							fTn := Interfacex.Parameters.PID_Condenser_Temp.Ti,
//							fTv := Interfacex.Parameters.PID_Condenser_Temp.Td,
//							fTd := Interfacex.Parameters.PID_Condenser_Temp.Tn,
//							fCtrlOutput => Condenser_Temp.ControlSignal);
								 
	CASE LPHeater_Temp.Switch OF 
		 0: 
			  LPHeater_Temp.ControlSignal := LPHeater_Temp.Setpoint/100;
		 1: 
			  LPHeater_Temp_PID(fSetpointValue := LPHeater_Temp.Setpoint,
						fActualValue := Streams.InStream.LPHeater_Temp,
						bReset := NOT PnID.LPHeaterValve.Cmd OR LPHeater_Temp.ResetPid,
						fCtrlCycleTime := Interfacex.Parameters.SampleTime,
						fKp := Interfacex.Parameters.PID_LPHeater_Temp.Kp,
						fTn := Interfacex.Parameters.PID_LPHeater_Temp.Ti,
						fTv := Interfacex.Parameters.PID_LPHeater_Temp.Td,
						fTd := Interfacex.Parameters.PID_LPHeater_Temp.Tn,
						fCtrlOutput => LPHeater_Temp.ControlSignal);
	END_CASE
	
	CASE AirEjector_Temp.Switch OF
		0:
			 AirEjector_Temp.ControlSignal := AirEjector_Temp.Setpoint/100;
		1: 
			 AirEjector_Temp_PID(fSetpointValue := AirEjector_Temp.Setpoint,
							fActualValue := Streams.InStream.AirEjector_Temp,
							bReset := NOT PnID.AirEjectorValve.Cmd OR AirEjector_Temp.ResetPid,
							fCtrlCycleTime := Interfacex.Parameters.SampleTime,
							fKp := Interfacex.Parameters.PID_AirEjector_Temp.Kp,
							fTn := Interfacex.Parameters.PID_AirEjector_Temp.Ti,
							fTv := Interfacex.Parameters.PID_AirEjector_Temp.Td,
							fTd := Interfacex.Parameters.PID_AirEjector_Temp.Tn,
							fCtrlOutput => AirEjector_Temp.ControlSignal);
	END_CASE							 
				
	CASE HPHeater_Temp.Switch OF
		0: 
			 HPHeater_Temp.ControlSignal := HPHeater_Temp.Setpoint/100;
		1: 
			 HPHeater_Temp_PID(fSetpointValue := HPHeater_Temp.Setpoint,
							fActualValue := Streams.InStream.HPHeater_Temp,
							bReset := NOT PnID.HPHeaterValve.Cmd OR HPHeater_Temp.ResetPid,
							fCtrlCycleTime := Interfacex.Parameters.SampleTime,
							fKp := Interfacex.Parameters.PID_HPHeater_Temp.Kp,
							fTn := Interfacex.Parameters.PID_HPHeater_Temp.Ti,
							fTv := Interfacex.Parameters.PID_HPHeater_Temp.Td,
							fTd := Interfacex.Parameters.PID_HPHeater_Temp.Tn,
							fCtrlOutput => HPHeater_Temp.ControlSignal);
	END_CASE				 
	
	CASE Turbine_Speed.Switch OF
		0:
			 Turbine_Speed.ControlSignal := Turbine_Speed.Setpoint/100;
		1: 
			 Turbine_Speed_PID(fSetpointValue := Turbine_Speed.Setpoint,
							fActualValue := Streams.InStream.Turbine_Rotation,
							bReset := NOT PnID.TurbineValve.Cmd OR Turbine_Speed.ResetPid,
							fCtrlCycleTime := Interfacex.Parameters.SampleTime,
							fKp := Interfacex.Parameters.PID_Turbine_Speed.Kp,
							fTn := Interfacex.Parameters.PID_Turbine_Speed.Ti,
							fTv := Interfacex.Parameters.PID_Turbine_Speed.Td,
							fTd := Interfacex.Parameters.PID_Turbine_Speed.Tn,
							fCtrlOutput => Turbine_Speed.ControlSignal);
	END_CASE
	
	Boiler_Temp_PID(fSetpointValue := Boiler_Temp.Setpoint,
							fActualValue := Streams.InStream.Boiler_Temp,
							bReset := NOT (PnID.ForceFan1.Cmd AND PnID.ForceFan2.Cmd AND PnID.ForceFan3.Cmd) OR Boiler_Temp.ResetPid,
							fCtrlCycleTime := Interfacex.Parameters.SampleTime,
							fKp := Interfacex.Parameters.PID_Boiler_Temp.Kp,
							fTn := Interfacex.Parameters.PID_Boiler_Temp.Ti,
							fTv := Interfacex.Parameters.PID_Boiler_Temp.Td,
							fTd := Interfacex.Parameters.PID_Boiler_Temp.Tn,
							fCtrlOutput => Boiler_Temp.ControlSignal);
							 
//END_IF
//Catch trigger of manual to automatic
CondensePump_Press_Trig(CLK := (PnID.CondensePump.Mode = aE_Mode.Auto));
SupplyPump_Press_Trig(CLK := (PnID.SupplyPump.Mode = aE_Mode.Auto));
//Condenser_Temp_Trig(CLK := (PnID.CircularPump.Mode = aE_Mode.Auto));
LPHeater_Temp_Trig(CLK := (PnID.LPHeaterValve.Mode = aE_Mode.Auto));
AirEjector_Temp_Trig(CLK := (PnID.AirEjectorValve.Mode = aE_Mode.Auto));
HPHeater_Temp_Trig(CLK := (PnID.HPHeaterValve.Mode = aE_Mode.Auto));
Turbine_Speed_Trig(CLK := (PnID.TurbineValve.Mode = aE_Mode.Auto));
Boiler_Temp_Trig(CLK := (PnID.ForceFan1.Mode = aE_Mode.Auto));

IF PnID.CondensePump.Mode = aE_Mode.Manual THEN
	CondensePump_Press.ResetPid := TRUE;
END_IF
IF PnID.SupplyPump.Mode = aE_Mode.Manual THEN
	SupplyPump_Press.ResetPid := TRUE;
END_IF
//IF PnID.CircularPump.Mode = aE_Mode.Manual THEN
//	Condenser_Temp.ResetPid := TRUE;
//END_IF
IF PnID.LPHeaterValve.Mode = aE_Mode.Manual THEN
	LPHeater_Temp.ResetPid := TRUE;
END_IF
IF PnID.AirEjectorValve.Mode = aE_Mode.Manual THEN
	AirEjector_Temp.ResetPid := TRUE;
END_IF
IF PnID.HPHeaterValve.Mode = aE_Mode.Manual THEN
	HPHeater_Temp.ResetPid := TRUE;
END_IF
IF PnID.TurbineValve.Mode = aE_Mode.Manual THEN
	Turbine_Speed.ResetPid := TRUE;
END_IF
IF PnID.ForceFan1.Mode = aE_Mode.Manual THEN
	Boiler_Temp.ResetPid := TRUE;
END_IF

IF CondensePump_Press_Trig.Q THEN
	CondensePump_Press.ResetPid := FALSE;
END_IF
IF SupplyPump_Press_Trig.Q THEN
	SupplyPump_Press.ResetPid := FALSE;
END_IF
//IF Condenser_Temp_Trig.Q THEN
//	Condenser_Temp.ResetPid := FALSE;
//END_IF
IF LPHeater_Temp_Trig.Q THEN
	LPHeater_Temp.ResetPid := FALSE;
END_IF
IF AirEjector_Temp_Trig.Q THEN
	AirEjector_Temp.ResetPid := FALSE;
END_IF
IF HPHeater_Temp_Trig.Q THEN
	HPHeater_Temp.ResetPid := FALSE;
END_IF
IF Turbine_Speed_Trig.Q THEN
	Turbine_Speed.ResetPid := FALSE;
END_IF
IF Boiler_Temp_Trig.Q THEN
	Boiler_Temp.ResetPid := FALSE;
END_IF
{endregion}

ACTION LockAllPidControllers:
CondensePump_Press.ResetPid := TRUE;
SupplyPump_Press.ResetPid := TRUE;
//Condenser_Temp.ResetPid := TRUE;
LPHeater_Temp.ResetPid := TRUE;
AirEjector_Temp.ResetPid := TRUE;
HPHeater_Temp.ResetPid := TRUE;
Turbine_Speed.ResetPid := TRUE;
Boiler_Temp.ResetPid := TRUE;
END_ACTION

ACTION Reset_StartAllComponents:
//Clear all start flags of components
CondensePump_Press.Start := FALSE;
SupplyPump_Press.Start := FALSE;
Condenser_Temp.Start := FALSE;
InterTank_Level.Start:= FALSE;
LPHeater_Temp.Start := FALSE;
AirEjector_Temp.Start := FALSE;
HPHeater_Temp.Start := FALSE;
Turbine_Speed.Start := FALSE;
Boiler_Temp.Start := FALSE;
END_ACTION

ACTION Reset_StopAllComponents:
//Reset all components
CondensePump_Press.Stop := FALSE;
SupplyPump_Press.Stop := FALSE;
Condenser_Temp.Stop := FALSE;
InterTank_Level.Stop := FALSE;
LPHeater_Temp.Stop := FALSE;
AirEjector_Temp.Stop := FALSE;
HPHeater_Temp.Stop := FALSE;
Turbine_Speed.Stop := FALSE;
Boiler_Temp.Stop := FALSE;
END_ACTION

ACTION ResetAllPidControllers:
//Reset all PID Controllers
CondensePump_Press_PID(bReset := TRUE);
SupplyPump_Press_PID(bReset := TRUE);
//Condenser_Temp_PID(bReset := TRUE);
LPHeater_Temp_PID(bReset := TRUE);
AirEjector_Temp_PID(bReset := TRUE);
HPHeater_Temp_PID(bReset := TRUE);
Turbine_Speed_PID(bReset := TRUE);
Boiler_Temp_PID(bReset := TRUE);
END_ACTION

ACTION StartAllComponents:
//Start all components
CondensePump_Press.Start := TRUE;
SupplyPump_Press.Start := TRUE;
//Condenser_Temp.Start := TRUE;
//InterTank_Level.Start := TRUE;
LPHeater_Temp.Start := TRUE;
AirEjector_Temp.Start := TRUE;
HPHeater_Temp.Start := TRUE;
Turbine_Speed.Start := TRUE;
Boiler_Temp.Start := TRUE;
END_ACTION

ACTION StopAllComponents:
//Stop all components
CondensePump_Press.Stop := TRUE;
SupplyPump_Press.Stop := TRUE;
Condenser_Temp.Stop := TRUE;
InterTank_Level.Stop := TRUE;
LPHeater_Temp.Stop := TRUE;
AirEjector_Temp.Stop := TRUE;
HPHeater_Temp.Stop := TRUE;
Turbine_Speed.Stop := TRUE;
Boiler_Temp.Stop := TRUE;
END_ACTION

ACTION UnlockAllPidControllers:
CondensePump_Press.ResetPid := FALSE;
SupplyPump_Press.ResetPid := FALSE;
//Condenser_Temp.ResetPid := FALSE;
LPHeater_Temp.ResetPid := FALSE;
AirEjector_Temp.ResetPid := FALSE;
HPHeater_Temp.ResetPid := FALSE;
Turbine_Speed.ResetPid := FALSE;
Boiler_Temp.ResetPid := FALSE;
END_ACTION

END_PROGRAM

// ---- POUs/PnID.TcPOU
PROGRAM PnID
VAR_INPUT
	CircularPumpFlow AT %I*: INT;
	bHI AT %I*: BOOL;
	bLO AT %I*: BOOL;
END_VAR
VAR_OUTPUT
	bMotor1 AT %Q*: BOOL;
	bMotor2 AT %Q*: BOOL;
END_VAR
VAR
	ForceFan1: aFb_Motor;
	ForceFan2: aFb_Motor;
	ForceFan3: aFb_Motor;
	CondensePump: aFb_Motor;
	SupplyPump: aFb_Motor;
	CircularPump: aFb_Motor;
	InterPump: aFb_Motor;
	LPHeaterValve: aFb_Valve;
	AirEjectorValve: aFb_Valve;
	HPHeaterValve: aFb_Valve;
	TurbineValve: aFb_Valve;
	
	CirPumpFlowT: INT;
	temp: REAL;
END_VAR

//Control all components in the P&ID 

//Resolve Flow Sensor
CirPumpFlowT:= CircularPumpFlow;
temp := (INT_TO_REAL(CirPumpFlowT) - 630)*0.0006;
IF temp < 0 THEN
	Streams.OutStream.CircularPump_OutFlow := 0;
ELSE
	Streams.OutStream.CircularPump_OutFlow := temp;
END_IF

//Pumps
{region "Condense Pump"}
CondensePump(RunCondition := AutoControl.CondensePump_Press.Start,
				StopCondition := AutoControl.CondensePump_Press.Stop,
				SpeedCondition := AutoControl.CondensePump_Press.ControlSignal,
				RunFeedback := CondensePump.Cmd,
				Maxspeed := Interfacex.Parameters.MaxSpeed_CondensePump,//.MaxSpeed_CondensePump,
				ActualSpeed := Streams.InStream.CondensePump_Speed ,
				Speed => Streams.OutStream.CondensePump_SetSpeed,
				DisplayName := 'Condense Pump');
{endregion}
{region "Supply Pump"}
SupplyPump(RunCondition := AutoControl.SupplyPump_Press.Start,
				StopCondition := AutoControl.SupplyPump_Press.Stop,
				SpeedCondition := AutoControl.SupplyPump_Press.ControlSignal,
				RunFeedback := SupplyPump.Cmd,
				Maxspeed := Interfacex.Parameters.MaxSpeed_SupplyPump,
				ActualSpeed := Streams.InStream.SupplyPump_Speed,
				Speed => Streams.OutStream.SupplyPump_SetSpeed,
				DisplayName := 'Supply Pump');
{endregion}
	 
{region "Circular Pump"}
CircularPump(RunCondition := AutoControl.Condenser_Temp.Start,
				StopCondition := AutoControl.Condenser_Temp.Stop,
				SpeedCondition := Interfacex.Parameters.MaxSpeed_CircularPump,
				RunFeedback := CircularPump.Cmd,
				Maxspeed := Interfacex.Parameters.MaxSpeed_CircularPump,
				ActualSpeed := CircularPump.Speed,
				Cmd => bMotor2,
				DisplayName := 'Circular Pump');
{endregion}
	 
{region 'Intermediate Pump'}
InterPump(RunCondition := AutoControl.InterTank_Level.Start,
				StopCondition := AutoControl.InterTank_Level.Stop,
				SpeedCondition := Interfacex.Parameters.MaxSpeed_InterPump,
				RunFeedback := InterPump.Cmd,
				Maxspeed := Interfacex.Parameters.MaxSpeed_InterPump,
				ActualSpeed := InterPump.Speed,
				Cmd => bMotor1,
				DisplayName := 'Intermediate Pump');
{endregion}


//Valves
{region "Low Pressure Heater Valve"}
LPHeaterValve(RunCondition := AutoControl.LPHeater_Temp.Start,
				StopCondition := AutoControl.LPHeater_Temp.Stop,
				PercentCondition := AutoControl.LPHeater_Temp.ControlSignal,
				RunFeedback := LPHeaterValve.Cmd,
				OpenPercent => Streams.OutStream.LPHeaterValve_SetPercent,
				DisplayName := 'Low Pressure Heater Valve');
{endregion}
	 
{region "Deaerator"}
AirEjectorValve(RunCondition := AutoControl.AirEjector_Temp.Start,
				StopCondition := AutoControl.AirEjector_Temp.Stop,
				PercentCondition := AutoControl.AirEjector_Temp.ControlSignal,
				RunFeedback := AirEjectorValve.Cmd,
				OpenPercent => Streams.OutStream.AirEjectorValve_SetPercent,
				DisplayName := 'Deaerator Valve');
{endregion}
{region "High Pressure Heater Valve"}
HPHeaterValve(RunCondition := AutoControl.HPHeater_Temp.Start,
				StopCondition := AutoControl.HPHeater_Temp.Stop,
				PercentCondition := AutoControl.HPHeater_Temp.ControlSignal,
				RunFeedback := HPHeaterValve.Cmd,
				OpenPercent => Streams.OutStream.HPHeaterValve_SetPercent,
				DisplayName := 'High Pressure Heater Valve');
{endregion}
{region "Turbine Valve"}
TurbineValve(RunCondition := AutoControl.Turbine_Speed.Start,
				StopCondition := AutoControl.Turbine_Speed.Stop,
				PercentCondition := AutoControl.Turbine_Speed.ControlSignal,
				RunFeedback := TurbineValve.Cmd,
				OpenPercent => Streams.OutStream.TurbineValve_SetPercent,
				DisplayName := 'Turbine Valve');
{endregion}


//Fans
{region "ForceFan1"}
ForceFan1(RunCondition := AutoControl.Boiler_Temp.Start,
				StopCondition := AutoControl.Boiler_Temp.Stop,
				SpeedCondition := AutoControl.Boiler_Temp.ControlSignal,
				RunFeedback := ForceFan1.Cmd,
				Maxspeed := Interfacex.Parameters.MaxSpeed_ForceFan1,
				ActualSpeed := Streams.InStream.ForceFan1_Speed,
				Speed => Streams.OutStream.ForceFan1_SetSpeed,
				DisplayName := 'Force Fan 1');
{endregion}
	 
{region "ForceFan2"}
ForceFan2(RunCondition := AutoControl.Boiler_Temp.Start,
				StopCondition := AutoControl.Boiler_Temp.Stop,
				SpeedCondition := AutoControl.Boiler_Temp.ControlSignal,
				RunFeedback := ForceFan2.Cmd,
				Maxspeed := Interfacex.Parameters.MaxSpeed_ForceFan2,
				ActualSpeed := Streams.InStream.ForceFan2_Speed,
				Speed => Streams.OutStream.ForceFan2_SetSpeed,
				DisplayName := 'Force Fan 2');
{endregion}
{region "ForceFan3"}
ForceFan3(RunCondition := AutoControl.Boiler_Temp.Start,
				StopCondition := AutoControl.Boiler_Temp.Stop,
				SpeedCondition := AutoControl.Boiler_Temp.ControlSignal,
				RunFeedback := ForceFan3.Cmd,
				Maxspeed := Interfacex.Parameters.MaxSpeed_ForceFan3,
				ActualSpeed := Streams.InStream.ForceFan3_Speed,
				Speed => Streams.OutStream.ForceFan3_SetSpeed,
				DisplayName := 'Force Fan 3');
{endregion}

END_PROGRAM

// ---- POUs/FB/aFb_Motor.TcPOU
FUNCTION_BLOCK aFb_Motor
VAR_INPUT
	Mode: aE_Mode := aE_Mode.Auto;
	
	//Manual
	Start: BOOL;
	Stop: BOOL;
	SetSpeed: REAL;
	Reset1: BOOL;
	
	//Auto
	RunCondition: BOOL;
	StopCondition: BOOL;
	SpeedCondition: REAL;
	
	//Others
	RunFeedback: BOOL;
	Interlock: BOOL;
	Maxspeed: REAL:= 1500;
	ActualSpeed: REAL;
	{attribute 'hide'}
	DisplayName: STRING[20];
END_VAR
VAR_OUTPUT
	Cmd: BOOL;
	Fault: BOOL;
	State: aE_State;
	Speed: REAL;
	Runtime: UDINT := 0;
	AccRuntime: UDINT := 0;
END_VAR
VAR
	{attribute 'hide'}
	fbTon: TON;
	{attribute 'hide'}
	fbTRuntime: TON;
	
	{attribute 'hide'}
	fbSource: FB_TcSourceInfo;
	{attribute 'hide'}
	fbMesModeMan: FB_TcMessage;
	{attribute 'hide'}
	fbMesModeAuto: FB_TcMessage;
	{attribute 'hide'}
	fbMesModeServ: FB_TcMessage;
	{attribute 'hide'}
	fbMesStart: FB_TcMessage;
	{attribute 'hide'}
	fbMesStop: FB_TcMessage;
	{attribute 'hide'}
	fbMesReset: FB_TcMessage;
	{attribute 'hide'}
	fbMesFault: FB_TcMessage;
	
	{attribute 'hide'}
	bFirstScan: BOOL := TRUE;
	{attribute 'hide'}
	trigModeMan: R_TRIG;
	{attribute 'hide'}
	trigModeAuto: R_TRIG;
	{attribute 'hide'}
	trigModeServ: R_TRIG;
	{attribute 'hide'}
	trigStart: R_TRIG;
	{attribute 'hide'}
	trigStop: R_TRIG;
	{attribute 'hide'}
	trigReset: R_TRIG;
	{attribute 'hide'}
	trigFault: R_TRIG;
	
END_VAR

IF bFirstScan THEN
	bFirstScan := FALSE;
	fbSource.sName := DisplayName;
	fbMesModeMan.CreateEx(TC_Events.ComponentEvent.ModeManual, fbSource);
	fbMesModeAuto.CreateEx(TC_Events.ComponentEvent.ModeAutomatic, fbSource);
	fbMesModeServ.CreateEx(TC_Events.ComponentEvent.ModeService, fbSource);
	fbMesStart.CreateEx(TC_Events.ComponentEvent.Started, fbSource);
	fbMesStop.CreateEx(TC_Events.ComponentEvent.Stopped, fbSource);
	fbMesReset.CreateEx(TC_Events.ComponentEvent.Resetted, fbSource);
	fbMesFault.CreateEx(TC_Events.ComponentEvent.Fault, fbSource);
END_IF

CASE Mode OF 
	aE_Mode.Manual: 
		Cmd := (Cmd OR Start) AND NOT Stop AND NOT Fault AND NOT Interlock;
		IF Cmd THEN
			State := aE_State.ManRun;
		ELSE
			State := aE_State.ManStop;
		END_IF
	aE_Mode.Auto:
		Cmd := (Cmd OR RunCondition) AND NOT StopCondition AND NOT Fault AND NOT Interlock;
		State := aE_State.Auto;
	aE_Mode.Service:
		Cmd := (Cmd OR Start) AND NOT Stop AND NOT Fault;
		IF Cmd THEN
			State := aE_State.ManRun;
		ELSE
			State := aE_State.ManStop;
		END_IF
END_CASE

IF Cmd THEN
	IF Mode = aE_Mode.Auto THEN
		Speed := LIMIT(-Maxspeed, SpeedCondition, Maxspeed);
	ELSE
		Speed := LIMIT(-Maxspeed, SetSpeed, Maxspeed);
	END_IF
ELSE 
	Speed:= 0;
END_IF

fbTon(IN := Cmd, PT := T#5S);
IF fbTon.Q AND NOT RunFeedback THEN
	Fault := TRUE;
	State := aE_State.Fault;
END_IF

IF Reset1 THEN
	Fault := FALSE;
END_IF

IF Cmd THEN
	fbTRuntime(IN := NOT fbTRuntime.Q, PT:= T#1S);
	IF fbTRuntime.Q THEN
		Runtime:= Runtime + 1;
		AccRuntime := AccRuntime + 1;
	END_IF
ELSE
	Runtime:= 0;
END_IF

trigModeMan(CLK:= (Mode = aE_Mode.Manual));
trigModeAuto(CLK:= (Mode = aE_Mode.Auto));
trigModeServ(CLK:= (Mode = aE_Mode.Service));
trigStart(CLK:= Start);
trigStop(CLK := Stop);
trigReset(CLK := Reset1);
trigFault(CLK := Fault);

IF trigModeMan.Q THEN
	fbMesModeMan.Send(0);
END_IF
IF trigModeAuto.Q THEN
	fbMesModeAuto.Send(0);
END_IF
IF trigModeServ.Q THEN
	fbMesModeServ.Send(0);
END_IF
IF trigStart.Q THEN
	fbMesStart.Send(0);
END_IF
IF trigStop.Q THEN
	fbMesStop.Send(0);
END_IF
IF trigReset.Q THEN
	fbMesReset.Send(0);
END_IF
IF trigFault.Q THEN
	fbMesFault.Send(0);
END_IF

END_FUNCTION_BLOCK

// ---- POUs/FB/aFB_Valve.TcPOU
FUNCTION_BLOCK aFb_Valve
VAR_INPUT
	Mode: aE_Mode := aE_Mode.Auto;
	
	//Manual
	Start: BOOL;
	Stop: BOOL;
	SetPercent: REAL;
	Reset1: BOOL;
	
	//Auto
	RunCondition: BOOL;
	StopCondition: BOOL;
	PercentCondition: REAL;
	
	//Others
	RunFeedback: BOOL;
	Interlock: BOOL;
	{attribute 'hide'}
	DisplayName: STRING[30];
END_VAR
VAR_OUTPUT
	Cmd: BOOL;
	Fault: BOOL;
	State: aE_State;
	OpenPercent: REAL;
	Runtime: UDINT := 0;
	AccRuntime: UDINT := 0;
END_VAR
VAR
	{attribute 'hide'}
	fbTon: TON;
	{attribute 'hide'}
	fbTRuntime: TON;	
	
	{attribute 'hide'}
	fbSource: FB_TcSourceInfo;
	{attribute 'hide'}
	fbMesModeMan: FB_TcMessage;
	{attribute 'hide'}
	fbMesModeAuto: FB_TcMessage;
	{attribute 'hide'}
	fbMesModeServ: FB_TcMessage;
	{attribute 'hide'}
	fbMesStart: FB_TcMessage;
	{attribute 'hide'}
	fbMesStop: FB_TcMessage;
	{attribute 'hide'}
	fbMesReset: FB_TcMessage;
	{attribute 'hide'}
	fbMesFault: FB_TcMessage;
	
	{attribute 'hide'}
	bFirstScan: BOOL := TRUE;
	{attribute 'hide'}
	trigModeMan: R_TRIG;
	{attribute 'hide'}
	trigModeAuto: R_TRIG;
	{attribute 'hide'}
	trigModeServ: R_TRIG;
	{attribute 'hide'}
	trigStart: R_TRIG;
	{attribute 'hide'}
	trigStop: R_TRIG;
	{attribute 'hide'}
	trigReset: R_TRIG;
	{attribute 'hide'}
	trigFault: R_TRIG;

END_VAR

IF bFirstScan THEN
	bFirstScan := FALSE;
	fbSource.sName := DisplayName;
	fbMesModeMan.CreateEx(TC_Events.ComponentEvent.ModeManual, fbSource);
	fbMesModeAuto.CreateEx(TC_Events.ComponentEvent.ModeAutomatic, fbSource);
	fbMesModeServ.CreateEx(TC_Events.ComponentEvent.ModeService, fbSource);
	fbMesStart.CreateEx(TC_Events.ComponentEvent.Started, fbSource);
	fbMesStop.CreateEx(TC_Events.ComponentEvent.Stopped, fbSource);
	fbMesReset.CreateEx(TC_Events.ComponentEvent.Resetted, fbSource);
	fbMesFault.CreateEx(TC_Events.ComponentEvent.Fault, fbSource);
END_IF

CASE Mode OF 
	aE_Mode.Manual: 
		Cmd := (Cmd OR Start) AND NOT Stop AND NOT Fault AND NOT Interlock;
		IF Cmd THEN
			State := aE_State.ManRun;
		ELSE
			State := aE_State.ManStop;
		END_IF
	aE_Mode.Auto:
		Cmd := (Cmd OR RunCondition) AND NOT StopCondition AND NOT Fault AND NOT Interlock;
		State := aE_State.Auto;
	aE_Mode.Service:
		Cmd := (Cmd OR Start) AND NOT Stop AND NOT Fault;
		IF Cmd THEN
			State := aE_State.ManRun;
		ELSE
			State := aE_State.ManStop;
		END_IF
END_CASE

IF Cmd THEN
	IF Mode = aE_Mode.Auto THEN
		OpenPercent := LIMIT( 0, PercentCondition, 1);
	ELSE
		OpenPercent := LIMIT( 0, SetPercent, 1);
	END_IF
ELSE 
	OpenPercent:= 0;
END_IF

fbTon(IN := Cmd, PT := T#3S);
IF fbTon.Q AND NOT RunFeedback THEN
	Fault := TRUE;
	State := aE_State.Fault;
END_IF

IF Reset1 THEN
	Fault := FALSE;
END_IF

IF Cmd THEN
	fbTRuntime(IN := NOT fbTRuntime.Q, PT:= T#1S);
	IF fbTRuntime.Q THEN
		Runtime:= Runtime + 1;
		AccRuntime := AccRuntime + 1;
	END_IF
ELSE
	Runtime:= 0;
END_IF

trigModeMan(CLK:= (Mode = aE_Mode.Manual));
trigModeAuto(CLK:= (Mode = aE_Mode.Auto));
trigModeServ(CLK:= (Mode = aE_Mode.Service));
trigStart(CLK:= Start);
trigStop(CLK := Stop);
trigReset(CLK := Reset1);
trigFault(CLK := Fault);

IF trigModeMan.Q THEN
	fbMesModeMan.Send(0);
END_IF
IF trigModeAuto.Q THEN
	fbMesModeAuto.Send(0);
END_IF
IF trigModeServ.Q THEN
	fbMesModeServ.Send(0);
END_IF
IF trigStart.Q THEN
	fbMesStart.Send(0);
END_IF
IF trigStop.Q THEN
	fbMesStop.Send(0);
END_IF
IF trigReset.Q THEN
	fbMesReset.Send(0);
END_IF
IF trigFault.Q THEN
	fbMesFault.Send(0);
END_IF

END_FUNCTION_BLOCK

// ---- POUs/AlarmManagement.TcPOU
PROGRAM AlarmManagement
VAR
{region 'Process Control Message'}
	bFirstScan: BOOL := TRUE;
	fbSource: FB_TcSourceInfo;
	
	fbMesInitialized: FB_TcMessage;
	fbMesEnabled: FB_TcMessage;
	fbMesStarting: FB_TcMessage;
	fbMesStarted: FB_TcMessage;
	fbMesSteadyState: FB_TcMessage;
	fbMesStopping: FB_TcMessage;
	fbMesStopped: FB_TcMessage;
	fbMesDisabled: FB_TcMessage;
	fbMesEmergency: FB_TcMessage;
	fbMesErrorEmergency: FB_TcMessage;
	fbMesResetted: FB_TcMessage;
	
	trigInitialized: F_TRIG;
	trigEnabled: F_TRIG;
	trigStarting: R_TRIG;
	trigStarted: F_TRIG;
	trigSteadyState: R_TRIG;
	trigStopping: R_TRIG;
	trigStopped: F_TRIG;
	trigDisabled: F_TRIG;
	trigEmergency: R_TRIG;
	trigErrorEmergency: R_TRIG;
	trigResetted: F_TRIG;
{endregion}
	
{region 'Process Alarm'}
	bFirstScan2: BOOL := TRUE;
	fbSLPHeaterTemp: FB_TcSourceInfo;
	fbSLPHeaterPress: FB_TcSourceInfo;
	fbSDeaeratorTemp: FB_TcSourceInfo;
	fbSHPHeaterTemp: FB_TcSourceInfo;
	fbSHPHeaterPress: FB_TcSourceInfo;
	fbSBoilerTemp: FB_TcSourceInfo;
	fbSCondenserTemp: FB_TcSourceInfo;
	fbSTurbineTemp: FB_TcSourceInfo;
	fbSTurbinePress: FB_TcSourceInfo;
	fbSTurbineRotation: FB_TcSourceInfo;
	
	fbAlLPHeaterTempHIHI: FB_TcAlarm;
	fbAlLPHeaterTempHI: FB_TcAlarm;
	fbAlLPHeaterTempLO: FB_TcAlarm;
	fbAlLPHeaterTempLOLO: FB_TcAlarm;
	fbAlLPHeaterPressHIHI: FB_TcAlarm;
	fbAlLPHeaterPressHI: FB_TcAlarm;
	fbAlLPHeaterPressLO: FB_TcAlarm;
	fbAlLPHeaterPressLOLO: FB_TcAlarm;
	fbAlDeaeratorTempHIHI: FB_TcAlarm;
	fbAlDeaeratorTempHI: FB_TcAlarm;
	fbAlDeaeratorTempLO: FB_TcAlarm;
	fbAlDeaeratorTempLOLO: FB_TcAlarm;
	fbAlHPHeaterTempHIHI: FB_TcAlarm;
	fbAlHPHeaterTempHI: FB_TcAlarm;
	fbAlHPHeaterTempLO: FB_TcAlarm;
	fbAlHPHeaterTempLOLO: FB_TcAlarm;
	fbAlHPHeaterPressHIHI: FB_TcAlarm;
	fbAlHPHeaterPressHI: FB_TcAlarm;
	fbAlHPHeaterPressLO: FB_TcAlarm;
	fbAlHPHeaterPressLOLO: FB_TcAlarm;
	fbAlBoilerTempHIHI: FB_TcAlarm;
	fbAlBoilerTempHI: FB_TcAlarm;
	fbAlBoilerTempLO: FB_TcAlarm;
	fbAlBoilerTempLOLO: FB_TcAlarm;
	fbAlCondenserTempHIHI: FB_TcAlarm;
	fbAlCondenserTempHI: FB_TcAlarm;
	fbAlCondenserTempLO: FB_TcAlarm;
	fbAlCondenserTempLOLO: FB_TcAlarm;
	fbAlTurbineTempHIHI: FB_TcAlarm;
	fbAlTurbineTempHI: FB_TcAlarm;
	fbAlTurbineTempLO: FB_TcAlarm;
	fbAlTurbineTempLOLO: FB_TcAlarm;
	fbAlTurbinePressHIHI: FB_TcAlarm;
	fbAlTurbinePressHI: FB_TcAlarm;
	fbAlTurbinePressLO: FB_TcAlarm;
	fbAlTurbinePressLOLO: FB_TcAlarm;
	fbAlTurbineRotationHIHI: FB_TcAlarm;
	fbAlTurbineRotationHI: FB_TcAlarm;
	fbAlTurbineRotationLO: FB_TcAlarm;
	fbAlTurbineRotationLOLO: FB_TcAlarm;

	trigRLPHTempHIHI: R_TRIG;
	trigRLPHTempHI: R_TRIG;
	trigRLPHTempLO: R_TRIG;
	trigRLPHTempLOLO: R_TRIG;
	trigRLPHPressHIHI: R_TRIG;
	trigRLPHPressHI: R_TRIG;
	trigRLPHPressLO: R_TRIG;
	trigRLPHPressLOLO: R_TRIG;
	trigRDeaerTempHIHI: R_TRIG;
	trigRDeaerTempHI: R_TRIG;
	trigRDeaerTempLO: R_TRIG;
	trigRDeaerTempLOLO: R_TRIG;
	trigRHPHTempHIHI: R_TRIG;
	trigRHPHTempHI: R_TRIG;
	trigRHPHTempLO: R_TRIG;
	trigRHPHTempLOLO: R_TRIG;
	trigRHPHPressHIHI: R_TRIG;
	trigRHPHPressHI: R_TRIG;
	trigRHPHPressLO: R_TRIG;
	trigRHPHPressLOLO: R_TRIG;
	trigRBoiTempHIHI: R_TRIG;
	trigRBoiTempHI: R_TRIG;
	trigRBoiTempLO: R_TRIG;
	trigRBoiTempLOLO: R_TRIG;
	trigRConTempHIHI: R_TRIG;
	trigRConTempHI: R_TRIG;
	trigRConTempLO: R_TRIG;
	trigRConTempLOLO: R_TRIG;
	trigRTurTempHIHI: R_TRIG;
	trigRTurTempHI: R_TRIG;
	trigRTurTempLO: R_TRIG;
	trigRTurTempLOLO: R_TRIG;
	trigRTurPressHIHI: R_TRIG;
	trigRTurPressHI: R_TRIG;
	trigRTurPressLO: R_TRIG;
	trigRTurPressLOLO: R_TRIG;
	trigRTurRotHIHI: R_TRIG;
	trigRTurRotHI: R_TRIG;
	trigRTurRotLO: R_TRIG;
	trigRTurRotLOLO: R_TRIG;
	
	trigFLPHTempHIHI: R_TRIG;
	trigFLPHTempHI: R_TRIG;
	trigFLPHTempLO: R_TRIG;
	trigFLPHTempLOLO: R_TRIG;
	trigFLPHPressHIHI: R_TRIG;
	trigFLPHPressHI: R_TRIG;
	trigFLPHPressLO: R_TRIG;
	trigFLPHPressLOLO: R_TRIG;
	trigFDeaerTempHIHI: R_TRIG;
	trigFDeaerTempHI: R_TRIG;
	trigFDeaerTempLO: R_TRIG;
	trigFDeaerTempLOLO: R_TRIG;
	trigFHPHTempHIHI: R_TRIG;
	trigFHPHTempHI: R_TRIG;
	trigFHPHTempLO: R_TRIG;
	trigFHPHTempLOLO: R_TRIG;
	trigFHPHPressHIHI: R_TRIG;
	trigFHPHPressHI: R_TRIG;
	trigFHPHPressLO: R_TRIG;
	trigFHPHPressLOLO: R_TRIG;
	trigFBoiTempHIHI: R_TRIG;
	trigFBoiTempHI: R_TRIG;
	trigFBoiTempLO: R_TRIG;
	trigFBoiTempLOLO: R_TRIG;
	trigFConTempHIHI: R_TRIG;
	trigFConTempHI: R_TRIG;
	trigFConTempLO: R_TRIG;
	trigFConTempLOLO: R_TRIG;
	trigFTurTempHIHI: R_TRIG;
	trigFTurTempHI: R_TRIG;
	trigFTurTempLO: R_TRIG;
	trigFTurTempLOLO: R_TRIG;
	trigFTurPressHIHI: R_TRIG;
	trigFTurPressHI: R_TRIG;
	trigFTurPressLO: R_TRIG;
	trigFTurPressLOLO: R_TRIG;
	trigFTurRotHIHI: R_TRIG;
	trigFTurRotHI: R_TRIG;
	trigFTurRotLO: R_TRIG;
	trigFTurRotLOLO: R_TRIG;
	
	bCfLPHeaterTempHIHI: BOOL;
	bCfLPHeaterTempHI: BOOL;
	bCfLPHeaterTempLO: BOOL;
	bCfLPHeaterTempLOLO: BOOL;
	bCfLPHeaterPressHIHI: BOOL;
	bCfLPHeaterPressHI: BOOL;
	bCfLPHeaterPressLO: BOOL;
	bCfLPHeaterPressLOLO: BOOL;
	bCfDeaeratorTempHIHI: BOOL;
	bCfDeaeratorTempHI: BOOL;
	bCfDeaeratorTempLO: BOOL;
	bCfDeaeratorTempLOLO: BOOL;
	bCfHPHeaterTempHIHI: BOOL;
	bCfHPHeaterTempHI: BOOL;
	bCfHPHeaterTempLO: BOOL;
	bCfHPHeaterTempLOLO: BOOL;
	bCfHPHeaterPressHIHI: BOOL;
	bCfHPHeaterPressHI: BOOL;
	bCfHPHeaterPressLO: BOOL;
	bCfHPHeaterPressLOLO: BOOL;
	bCfBoilerTempHIHI: BOOL;
	bCfBoilerTempHI: BOOL;
	bCfBoilerTempLO: BOOL;
	bCfBoilerTempLOLO: BOOL;
	bCfCondenserTempHIHI: BOOL;
	bCfCondenserTempHI: BOOL;
	bCfCondenserTempLO: BOOL;
	bCfCondenserTempLOLO: BOOL;
	bCfTurbineTempHIHI: BOOL;
	bCfTurbineTempHI: BOOL;
	bCfTurbineTempLO: BOOL;
	bCfTurbineTempLOLO: BOOL;
	bCfTurbinePressHIHI: BOOL;
	bCfTurbinePressHI: BOOL;
	bCfTurbinePressLO: BOOL;
	bCfTurbinePressLOLO: BOOL;
	bCfTurbineRotationHIHI: BOOL;
	bCfTurbineRotationHI: BOOL;
	bCfTurbineRotationLO: BOOL;
	bCfTurbineRotationLOLO: BOOL;
{endregion}

END_VAR

{region 'Process Control Message'}
IF bFirstScan THEN
	bFirstScan := FALSE;
	fbSource.sName := 'Process Controller';
	fbMesInitialized.CreateEx(TC_Events.ProcessEvent.Initialized, fbSource);
	fbMesEnabled.CreateEx(TC_Events.ProcessEvent.Enabled, fbSource);
	fbMesStarting.CreateEx(TC_Events.ProcessEvent.Starting, fbSource);
	fbMesStarted.CreateEx(TC_Events.ProcessEvent.Started, fbSource);
	fbMesSteadyState.CreateEx(TC_Events.ProcessEvent.SteadyState, fbSource);
	fbMesStopping.CreateEx(TC_Events.ProcessEvent.Stopping, fbSource);
	fbMesStopped.CreateEx(TC_Events.ProcessEvent.Stopped, fbSource);
	fbMesDisabled.CreateEx(TC_Events.ProcessEvent.Disabled, fbSource);
	fbMesEmergency.CreateEx(TC_Events.ProcessEvent.Emergency, fbSource);
	fbMesErrorEmergency.CreateEx(TC_Events.ProcessEvent.ErrorEmergency, fbSource);
	fbMesResetted.CreateEx(TC_Events.ProcessEvent.Resetted, fbSource);
END_IF

trigInitialized(CLK:= (AutoControl.ProcessState = aE_ProcessState.Init));
trigEnabled(CLK:= (AutoControl.ProcessState = aE_ProcessState.Enable));
trigStarting(CLK:= (AutoControl.ProcessState = aE_ProcessState.Start));
trigStarted(CLK:= (AutoControl.ProcessState = aE_ProcessState.Start));
trigSteadyState(CLK:= (AutoControl.ProcessState = aE_ProcessState.SteadyState));
trigStopping(CLK:= (AutoControl.ProcessState = aE_ProcessState.Stop));
trigStopped(CLK:= (AutoControl.ProcessState = aE_ProcessState.Stop));
trigDisabled(CLK:= (AutoControl.ProcessState = aE_ProcessState.Disable));
trigEmergency(CLK:= AutoControl.ProcessEmergency);
trigErrorEmergency(CLK:= (AutoControl.ProcessState = aE_ProcessState.Error));
trigResetted(CLK:= (AutoControl.ProcessState = aE_ProcessState.Reset));

IF trigInitialized.Q THEN
	fbMesInitialized.Send(0);
END_IF
IF trigEnabled.Q THEN
	fbMesEnabled.Send(0);
END_IF
IF trigStarting.Q THEN
	fbMesStarting.Send(0);
END_IF
IF trigStarted.Q THEN
	fbMesStarted.Send(0);
END_IF
IF trigSteadyState.Q THEN
	fbMesSteadyState.Send(0);
END_IF
IF trigStopping.Q THEN
	fbMesStopping.Send(0);
END_IF
IF trigStopped.Q THEN
	fbMesStopped.Send(0);
END_IF
IF trigDisabled.Q THEN
	fbMesDisabled.Send(0);
END_IF
IF trigEmergency.Q THEN
	fbMesEmergency.Send(0);
END_IF
IF trigErrorEmergency.Q THEN
	fbMesErrorEmergency.Send(0);
END_IF
IF trigResetted.Q THEN
	fbMesResetted.Send(0);
END_IF
{endregion}

{region 'Process Alarm'}

IF bFirstScan2 THEN
	bFirstScan2 := FALSE;
	fbSLPHeaterTemp.sName := 'LP Heater Temperature';
	fbSLPHeaterPress.sName := 'LP Heater Pressure';
	fbSDeaeratorTemp.sName := 'Deaerator Temperature';
	fbSHPHeaterTemp.sName := 'HP Heater Temperature';
	fbSHPHeaterPress.sName := 'HP Heater Pressure';
	fbSBoilerTemp.sName := 'Boiler Temperature';
	fbSCondenserTemp.sName := 'Condenser Temperature';
	fbSTurbineTemp.sName := 'Turbine Temperature';
	fbSTurbinePress.sName := 'Turbine Pressure';
	fbSTurbineRotation.sName := 'Turbine Speed';
	
	fbAlLPHeaterTempHIHI.CreateEx(TC_Events.AnalogAlarm.HiHi, TRUE,fbSLPHeaterTemp);
	fbAlLPHeaterTempHI.CreateEx(TC_Events.AnalogAlarm.Hi, TRUE,fbSLPHeaterTemp);
	fbAlLPHeaterTempLO.CreateEx(TC_Events.AnalogAlarm.Lo, TRUE,fbSLPHeaterTemp);
	fbAlLPHeaterTempLOLO.CreateEx(TC_Events.AnalogAlarm.LoLo, TRUE,fbSLPHeaterTemp);
	fbAlLPHeaterPressHIHI.CreateEx(TC_Events.AnalogAlarm.HiHi, TRUE,fbSLPHeaterPress);
	fbAlLPHeaterPressHI.CreateEx(TC_Events.AnalogAlarm.Hi, TRUE,fbSLPHeaterPress);
	fbAlLPHeaterPressLO.CreateEx(TC_Events.AnalogAlarm.Lo, TRUE,fbSLPHeaterPress);
	fbAlLPHeaterPressLOLO.CreateEx(TC_Events.AnalogAlarm.LoLo, TRUE,fbSLPHeaterPress);
	fbAlDeaeratorTempHIHI.CreateEx(TC_Events.AnalogAlarm.HiHi, TRUE,fbSDeaeratorTemp);
	fbAlDeaeratorTempHI.CreateEx(TC_Events.AnalogAlarm.Hi, TRUE,fbSDeaeratorTemp);
	fbAlDeaeratorTempLO.CreateEx(TC_Events.AnalogAlarm.Lo, TRUE,fbSDeaeratorTemp);
	fbAlDeaeratorTempLOLO.CreateEx(TC_Events.AnalogAlarm.LoLo, TRUE,fbSDeaeratorTemp);
	fbAlHPHeaterTempHIHI.CreateEx(TC_Events.AnalogAlarm.HiHi, TRUE,fbSHPHeaterTemp);
	fbAlHPHeaterTempHI.CreateEx(TC_Events.AnalogAlarm.Hi, TRUE,fbSHPHeaterTemp);
	fbAlHPHeaterTempLO.CreateEx(TC_Events.AnalogAlarm.Lo, TRUE,fbSHPHeaterTemp);
	fbAlHPHeaterTempLOLO.CreateEx(TC_Events.AnalogAlarm.LoLo, TRUE,fbSHPHeaterTemp);
	fbAlHPHeaterPressHIHI.CreateEx(TC_Events.AnalogAlarm.HiHi, TRUE,fbSHPHeaterPress);
	fbAlHPHeaterPressHI.CreateEx(TC_Events.AnalogAlarm.Hi, TRUE,fbSHPHeaterPress);
	fbAlHPHeaterPressLO.CreateEx(TC_Events.AnalogAlarm.Lo, TRUE,fbSHPHeaterPress);
	fbAlHPHeaterPressLOLO.CreateEx(TC_Events.AnalogAlarm.LoLo, TRUE,fbSHPHeaterPress);
	fbAlBoilerTempHIHI.CreateEx(TC_Events.AnalogAlarm.HiHi, TRUE,fbSBoilerTemp);
	fbAlBoilerTempHI.CreateEx(TC_Events.AnalogAlarm.Hi, TRUE,fbSBoilerTemp);
	fbAlBoilerTempLO.CreateEx(TC_Events.AnalogAlarm.Lo, TRUE,fbSBoilerTemp);
	fbAlBoilerTempLOLO.CreateEx(TC_Events.AnalogAlarm.LoLo, TRUE,fbSBoilerTemp);
	fbAlCondenserTempHIHI.CreateEx(TC_Events.AnalogAlarm.HiHi, TRUE,fbSCondenserTemp);
	fbAlCondenserTempHI.CreateEx(TC_Events.AnalogAlarm.Hi, TRUE,fbSCondenserTemp);
	fbAlCondenserTempLO.CreateEx(TC_Events.AnalogAlarm.Lo, TRUE,fbSCondenserTemp);
	fbAlCondenserTempLOLO.CreateEx(TC_Events.AnalogAlarm.LoLo, TRUE,fbSCondenserTemp);
	fbAlTurbineTempHIHI.CreateEx(TC_Events.AnalogAlarm.HiHi, TRUE,fbSTurbineTemp);
	fbAlTurbineTempHI.CreateEx(TC_Events.AnalogAlarm.Hi, TRUE,fbSTurbineTemp);
	fbAlTurbineTempLO.CreateEx(TC_Events.AnalogAlarm.Lo, TRUE,fbSTurbineTemp);
	fbAlTurbineTempLOLO.CreateEx(TC_Events.AnalogAlarm.LoLo, TRUE,fbSTurbineTemp);
	fbAlTurbinePressHIHI.CreateEx(TC_Events.AnalogAlarm.HiHi, TRUE,fbSTurbinePress);
	fbAlTurbinePressHI.CreateEx(TC_Events.AnalogAlarm.Hi, TRUE,fbSTurbinePress);
	fbAlTurbinePressLO.CreateEx(TC_Events.AnalogAlarm.Lo, TRUE,fbSTurbinePress);
	fbAlTurbinePressLOLO.CreateEx(TC_Events.AnalogAlarm.LoLo, TRUE,fbSTurbinePress);
	fbAlTurbineRotationHIHI.CreateEx(TC_Events.AnalogAlarm.HiHi, TRUE,fbSTurbineRotation);
	fbAlTurbineRotationHI.CreateEx(TC_Events.AnalogAlarm.Hi, TRUE,fbSTurbineRotation);
	fbAlTurbineRotationLO.CreateEx(TC_Events.AnalogAlarm.Lo, TRUE,fbSTurbineRotation);
	fbAlTurbineRotationLOLO.CreateEx(TC_Events.AnalogAlarm.LoLo, TRUE,fbSTurbineRotation);

END_IF

IF AutoControl.ProcessState = aE_ProcessState.SteadyState THEN	
	trigRLPHTempHIHI(CLK := (Streams.InStream.LPHeater_Temp > (AlarmLimit.alLPHeaterTemp.HIHI)));
	trigRLPHTempHI(CLK := (Streams.InStream.LPHeater_Temp > (AlarmLimit.alLPHeaterTemp.HI)));
	trigRLPHTempLO(CLK := (Streams.InStream.LPHeater_Temp < (AlarmLimit.alLPHeaterTemp.LO)));
	trigRLPHTempLOLO(CLK := (Streams.InStream.LPHeater_Temp < (AlarmLimit.alLPHeaterTemp.lolo)));
	trigRLPHPressHIHI(CLK := (Streams.InStream.LPHeater_Press > (AlarmLimit.alLPHeaterPress.HIHI)));
	trigRLPHPressHI(CLK := (Streams.InStream.LPHeater_Press > (AlarmLimit.alLPHeaterPress.HI)));
	trigRLPHPressLO(CLK := (Streams.InStream.LPHeater_Press < (AlarmLimit.alLPHeaterPress.lo)));
	trigRLPHPressLOLO(CLK := (Streams.InStream.LPHeater_Press < (AlarmLimit.alLPHeaterPress.LOLO)));
	trigRDeaerTempHIHI(CLK := (Streams.InStream.AirEjector_Temp > (AlarmLimit.alDeaeratorTemp.HIHI)));
	trigRDeaerTempHI(CLK := (Streams.InStream.AirEjector_Temp > (AlarmLimit.alDeaeratorTemp.HI)));
	trigRDeaerTempLO(CLK := (Streams.InStream.AirEjector_Temp < (AlarmLimit.alDeaeratorTemp.lo)));
	trigRDeaerTempLOLO(CLK := (Streams.InStream.AirEjector_Temp < (AlarmLimit.alDeaeratorTemp.LOLO)));
	trigRHPHTempHIHI(CLK := (Streams.InStream.HPHeater_Temp > (AlarmLimit.alHPHeaterTemp.HIHI)));
	trigRHPHTempHI(CLK := (Streams.InStream.HPHeater_Temp > (AlarmLimit.alHPHeaterTemp.HI)));
	trigRHPHTempLO(CLK := (Streams.InStream.HPHeater_Temp < (AlarmLimit.alHPHeaterTemp.LO)));
	trigRHPHTempLOLO(CLK := (Streams.InStream.HPHeater_Temp < (AlarmLimit.alHPHeaterTemp.LOLO)));
	trigRHPHPressHIHI(CLK := (Streams.InStream.HPHeater_Press > (AlarmLimit.alHPHeaterPress.HIHI)));
	trigRHPHPressHI(CLK := (Streams.InStream.HPHeater_Press > (AlarmLimit.alHPHeaterPress.HI)));
	trigRHPHPressLO(CLK := (Streams.InStream.HPHeater_Press < (AlarmLimit.alHPHeaterPress.LO)));
	trigRHPHPressLOLO(CLK := (Streams.InStream.HPHeater_Press < (AlarmLimit.alHPHeaterPress.LOLO)));
	trigRBoiTempHIHI(CLK := (Streams.InStream.Boiler_Temp > (AlarmLimit.alBoilerTemp.HIHI)));
	trigRBoiTempHI(CLK := (Streams.InStream.Boiler_Temp > (AlarmLimit.alBoilerTemp.HI)));
	trigRBoiTempLO(CLK := (Streams.InStream.Boiler_Temp < (AlarmLimit.alBoilerTemp.LO)));
	trigRBoiTempLOLO(CLK := (Streams.InStream.Boiler_Temp < (AlarmLimit.alBoilerTemp.LOLO)));
	trigRConTempHIHI(CLK := (Streams.InStream.Condenser_Temp > (AlarmLimit.alCondenserTemp.HIHI)));
	trigRConTempHI(CLK := (Streams.InStream.Condenser_Temp > (AlarmLimit.alCondenserTemp.HI)));
	trigRConTempLO(CLK := (Streams.InStream.Condenser_Temp < (AlarmLimit.alCondenserTemp.LO)));
	trigRConTempLOLO(CLK := (Streams.InStream.Condenser_Temp < (AlarmLimit.alCondenserTemp.LOLO)));
	trigRTurTempHIHI(CLK := (Streams.InStream.Turbine_OutTemp > (AlarmLimit.alTurbineTemp.HIHI)));
	trigRTurTempHI(CLK := (Streams.InStream.Turbine_OutTemp > (AlarmLimit.alTurbineTemp.HI)));
	trigRTurTempLO(CLK := (Streams.InStream.Turbine_OutTemp < (AlarmLimit.alTurbineTemp.LO)));
	trigRTurTempLOLO(CLK := (Streams.InStream.Turbine_OutTemp < (AlarmLimit.alTurbineTemp.LOLO)));
	trigRTurPressHIHI(CLK := (Streams.InStream.Turbine_OutPress > (AlarmLimit.alTurbinePress.HIHI)));
	trigRTurPressHI(CLK := (Streams.InStream.Turbine_OutPress > (AlarmLimit.alTurbinePress.HI)));
	trigRTurPressLO(CLK := (Streams.InStream.Turbine_OutPress < (AlarmLimit.alTurbinePress.LO)));
	trigRTurPressLOLO(CLK := (Streams.InStream.Turbine_OutPress < (AlarmLimit.alTurbinePress.LOLO)));
	trigRTurRotHIHI(CLK := (Streams.InStream.Turbine_Rotation > (AlarmLimit.alTurbineRotation.HIHI)));
	trigRTurRotHI(CLK := (Streams.InStream.Turbine_Rotation > (AlarmLimit.alTurbineRotation.HI)));
	trigRTurRotLO(CLK := (Streams.InStream.Turbine_Rotation < (AlarmLimit.alTurbineRotation.LO)));
	trigRTurRotLOLO(CLK := (Streams.InStream.Turbine_Rotation < (AlarmLimit.alTurbineRotation.LOLO)));
	
	trigFLPHTempHIHI(CLK := (Streams.InStream.LPHeater_Temp < (AlarmLimit.alLPHeaterTemp.HIHI - AlarmLimit.alLPHeaterTemp.Deadband)));
	trigFLPHTempHI(CLK := (Streams.InStream.LPHeater_Temp < (AlarmLimit.alLPHeaterTemp.HI - AlarmLimit.alLPHeaterTemp.Deadband)));
	trigFLPHTempLO(CLK := (Streams.InStream.LPHeater_Temp > (AlarmLimit.alLPHeaterTemp.LO - AlarmLimit.alLPHeaterTemp.Deadband)));
	trigFLPHTempLOLO(CLK := (Streams.InStream.LPHeater_Temp > (AlarmLimit.alLPHeaterTemp.LOLO - AlarmLimit.alLPHeaterTemp.Deadband)));
	trigFLPHPressHIHI(CLK := (Streams.InStream.LPHeater_Press < (AlarmLimit.alLPHeaterPress.HIHI - AlarmLimit.alLPHeaterPress.Deadband)));
	trigFLPHPressHI(CLK := (Streams.InStream.LPHeater_Press < (AlarmLimit.alLPHeaterPress.HI - AlarmLimit.alLPHeaterPress.Deadband)));
	trigFLPHPressLO(CLK := (Streams.InStream.LPHeater_Press > (AlarmLimit.alLPHeaterPress.LO - AlarmLimit.alLPHeaterPress.Deadband)));
	trigFLPHPressLOLO(CLK := (Streams.InStream.LPHeater_Press > (AlarmLimit.alLPHeaterPress.LOLO - AlarmLimit.alLPHeaterPress.Deadband)));
	trigFDeaerTempHIHI(CLK := (Streams.InStream.AirEjector_Temp < (AlarmLimit.alDeaeratorTemp.HIHI - AlarmLimit.alDeaeratorTemp.Deadband)));
	trigFDeaerTempHI(CLK := (Streams.InStream.AirEjector_Temp < (AlarmLimit.alDeaeratorTemp.HI - AlarmLimit.alDeaeratorTemp.Deadband)));
	trigFDeaerTempLO(CLK := (Streams.InStream.AirEjector_Temp > (AlarmLimit.alDeaeratorTemp.LO - AlarmLimit.alDeaeratorTemp.Deadband)));
	trigFDeaerTempLOLO(CLK := (Streams.InStream.AirEjector_Temp > (AlarmLimit.alDeaeratorTemp.LOLO - AlarmLimit.alDeaeratorTemp.Deadband)));
	trigFHPHTempHIHI(CLK := (Streams.InStream.HPHeater_Temp < (AlarmLimit.alHPHeaterTemp.HIHI - AlarmLimit.alHPHeaterTemp.Deadband)));
	trigFHPHTempHI(CLK := (Streams.InStream.HPHeater_Temp < (AlarmLimit.alHPHeaterTemp.HI - AlarmLimit.alHPHeaterTemp.Deadband)));
	trigFHPHTempLO(CLK := (Streams.InStream.HPHeater_Temp > (AlarmLimit.alHPHeaterTemp.LO - AlarmLimit.alHPHeaterTemp.Deadband)));
	trigFHPHTempLOLO(CLK := (Streams.InStream.HPHeater_Temp > (AlarmLimit.alHPHeaterTemp.LOLO - AlarmLimit.alHPHeaterTemp.Deadband)));
	trigFHPHPressHIHI(CLK := (Streams.InStream.HPHeater_Press < (AlarmLimit.alHPHeaterPress.HIHI - AlarmLimit.alHPHeaterPress.Deadband)));
	trigFHPHPressHI(CLK := (Streams.InStream.HPHeater_Press < (AlarmLimit.alHPHeaterPress.HI - AlarmLimit.alHPHeaterPress.Deadband)));
	trigFHPHPressLO(CLK := (Streams.InStream.HPHeater_Press > (AlarmLimit.alHPHeaterPress.LO - AlarmLimit.alHPHeaterPress.Deadband)));
	trigFHPHPressLOLO(CLK := (Streams.InStream.HPHeater_Press > (AlarmLimit.alHPHeaterPress.LOLO - AlarmLimit.alHPHeaterPress.Deadband)));
	trigFBoiTempHIHI(CLK := (Streams.InStream.Boiler_Temp < (AlarmLimit.alBoilerTemp.HIHI - AlarmLimit.alBoilerTemp.Deadband)));
	trigFBoiTempHI(CLK := (Streams.InStream.Boiler_Temp < (AlarmLimit.alBoilerTemp.HI - AlarmLimit.alBoilerTemp.Deadband)));
	trigFBoiTempLO(CLK := (Streams.InStream.Boiler_Temp > (AlarmLimit.alBoilerTemp.LO - AlarmLimit.alBoilerTemp.Deadband)));
	trigFBoiTempLOLO(CLK := (Streams.InStream.Boiler_Temp > (AlarmLimit.alBoilerTemp.LOLO - AlarmLimit.alBoilerTemp.Deadband)));
	trigFConTempHIHI(CLK := (Streams.InStream.Condenser_Temp < (AlarmLimit.alCondenserTemp.HIHI - AlarmLimit.alCondenserTemp.Deadband)));
	trigFConTempHI(CLK := (Streams.InStream.Condenser_Temp < (AlarmLimit.alCondenserTemp.HI - AlarmLimit.alCondenserTemp.Deadband)));
	trigFConTempLO(CLK := (Streams.InStream.Condenser_Temp > (AlarmLimit.alCondenserTemp.LO - AlarmLimit.alCondenserTemp.Deadband)));
	trigFConTempLOLO(CLK := (Streams.InStream.Condenser_Temp > (AlarmLimit.alCondenserTemp.LOLO - AlarmLimit.alCondenserTemp.Deadband)));
	trigFTurTempHIHI(CLK := (Streams.InStream.Turbine_OutTemp < (AlarmLimit.alTurbineTemp.HIHI - AlarmLimit.alTurbineTemp.Deadband)));
	trigFTurTempHI(CLK := (Streams.InStream.Turbine_OutTemp < (AlarmLimit.alTurbineTemp.HI - AlarmLimit.alTurbineTemp.Deadband)));
	trigFTurTempLO(CLK := (Streams.InStream.Turbine_OutTemp > (AlarmLimit.alTurbineTemp.LO - AlarmLimit.alTurbineTemp.Deadband)));
	trigFTurTempLOLO(CLK := (Streams.InStream.Turbine_OutTemp > (AlarmLimit.alTurbineTemp.LOLO - AlarmLimit.alTurbineTemp.Deadband)));
	trigFTurPressHIHI(CLK := (Streams.InStream.Turbine_OutPress < (AlarmLimit.alTurbinePress.HIHI - AlarmLimit.alTurbinePress.Deadband)));
	trigFTurPressHI(CLK := (Streams.InStream.Turbine_OutPress < (AlarmLimit.alTurbinePress.HI - AlarmLimit.alTurbinePress.Deadband)));
	trigFTurPressLO(CLK := (Streams.InStream.Turbine_OutPress > (AlarmLimit.alTurbinePress.LO - AlarmLimit.alTurbinePress.Deadband)));
	trigFTurPressLOLO(CLK := (Streams.InStream.Turbine_OutPress > (AlarmLimit.alTurbinePress.LOLO - AlarmLimit.alTurbinePress.Deadband)));
	trigFTurRotHIHI(CLK := (Streams.InStream.Turbine_Rotation < (AlarmLimit.alTurbineRotation.HIHI - AlarmLimit.alTurbineRotation.Deadband)));
	trigFTurRotHI(CLK := (Streams.InStream.Turbine_Rotation < (AlarmLimit.alTurbineRotation.HI - AlarmLimit.alTurbineRotation.Deadband)));
	trigFTurRotLO(CLK := (Streams.InStream.Turbine_Rotation > (AlarmLimit.alTurbineRotation.LO - AlarmLimit.alTurbineRotation.Deadband)));
	trigFTurRotLOLO(CLK := (Streams.InStream.Turbine_Rotation > (AlarmLimit.alTurbineRotation.LOLO - AlarmLimit.alTurbineRotation.Deadband)));

	IF trigRLPHTempHIHI.Q THEN
		fbAlLPHeaterTempHIHI.Raise(0);
	END_IF
	IF trigRLPHTempHI.Q THEN
		fbAlLPHeaterTempHI.Raise(0);
	END_IF
	IF trigRLPHTempLO.Q THEN
		fbAlLPHeaterTempLO.Raise(0);
	END_IF
	IF trigRLPHTempLOLO.Q THEN
		fbAlLPHeaterTempLOLO.Raise(0);
	END_IF
	IF trigRLPHPressHIHI.Q THEN
		fbAlLPHeaterPressHIHI.Raise(0);
	END_IF
	IF trigRLPHPressHI.Q THEN
		fbAlLPHeaterPressHI.Raise(0);
	END_IF
	IF trigRLPHPressLO.Q THEN
		fbAlLPHeaterPressLO.Raise(0);
	END_IF
	IF trigRLPHPressLOLO.Q THEN
		fbAlLPHeaterPressLOLO.Raise(0);
	END_IF
	IF trigRDeaerTempHIHI.Q THEN
		fbAlDeaeratorTempHIHI.Raise(0);
	END_IF
	IF trigRDeaerTempHI.Q THEN
		fbAlDeaeratorTempHI.Raise(0);
	END_IF
	IF trigRDeaerTempLO.Q THEN
		fbAlDeaeratorTempLO.Raise(0);
	END_IF
	IF trigRDeaerTempLOLO.Q THEN
		fbAlDeaeratorTempLOLO.Raise(0);
	END_IF
	IF trigRHPHTempHIHI.Q THEN
		fbAlHPHeaterTempHIHI.Raise(0);
	END_IF
	IF trigRHPHTempHI.Q THEN
		fbAlHPHeaterTempHI.Raise(0);
	END_IF
	IF trigRHPHTempLO.Q THEN
		fbAlHPHeaterTempLO.Raise(0);
	END_IF
	IF trigRHPHTempLOLO.Q THEN
		fbAlHPHeaterTempLOLO.Raise(0);
	END_IF
	IF trigRHPHPressHIHI.Q THEN
		fbAlHPHeaterPressHIHI.Raise(0);
	END_IF
	IF trigRHPHPressHI.Q THEN
		fbAlHPHeaterPressHI.Raise(0);
	END_IF
	IF trigRHPHPressLO.Q THEN
		fbAlHPHeaterPressLO.Raise(0);
	END_IF
	IF trigRHPHPressLOLO.Q THEN
		fbAlHPHeaterPressLOLO.Raise(0);
	END_IF
	IF trigRBoiTempHIHI.Q THEN
		fbAlBoilerTempHIHI.Raise(0);
	END_IF
	IF trigRBoiTempHI.Q THEN
		fbAlBoilerTempHI.Raise(0);
	END_IF
	IF trigRBoiTempLO.Q THEN
		fbAlBoilerTempLO.Raise(0);
	END_IF
	IF trigRBoiTempLOLO.Q THEN
		fbAlBoilerTempLOLO.Raise(0);
	END_IF
	IF trigRConTempHIHI.Q THEN
		fbAlCondenserTempHIHI.Raise(0);
	END_IF
	IF trigRConTempHI.Q THEN
		fbAlCondenserTempHI.Raise(0);
	END_IF
	IF trigRConTempLO.Q THEN
		fbAlCondenserTempLO.Raise(0);
	END_IF
	IF trigRConTempLOLO.Q THEN
		fbAlCondenserTempLOLO.Raise(0);
	END_IF
	IF trigRTurTempHIHI.Q THEN
		fbAlTurbineTempHIHI.Raise(0);
	END_IF
	IF trigRTurTempHI.Q THEN
		fbAlTurbineTempHI.Raise(0);
	END_IF
	IF trigRTurTempLO.Q THEN
		fbAlTurbineTempLO.Raise(0);
	END_IF
	IF trigRTurTempLOLO.Q THEN
		fbAlTurbineTempLOLO.Raise(0);
	END_IF
	IF trigRTurPressHIHI.Q THEN
		fbAlTurbinePressHIHI.Raise(0);
	END_IF
	IF trigRTurPressHI.Q THEN
		fbAlTurbinePressHI.Raise(0);
	END_IF
	IF trigRTurPressLO.Q THEN
		fbAlTurbinePressLO.Raise(0);
	END_IF
	IF trigRTurPressLOLO.Q THEN
		fbAlTurbinePressLOLO.Raise(0);
	END_IF
	IF trigRTurRotHIHI.Q THEN
		fbAlTurbineRotationHIHI.Raise(0);
	END_IF
	IF trigRTurRotHI.Q THEN
		fbAlTurbineRotationHI.Raise(0);
	END_IF
	IF trigRTurRotLO.Q THEN
		fbAlTurbineRotationLO.Raise(0);
	END_IF
	IF trigRTurRotLOLO.Q THEN
		fbAlTurbineRotationLOLO.Raise(0);
	END_IF

	IF trigFLPHTempHIHI.Q THEN
		fbAlLPHeaterTempHIHI.Clear(0, TRUE);
	END_IF
	IF trigFLPHTempHI.Q THEN
		fbAlLPHeaterTempHI.Clear(0, TRUE);
	END_IF
	IF trigFLPHTempLO.Q THEN
		fbAlLPHeaterTempLO.Clear(0, TRUE);
	END_IF
	IF trigFLPHTempLOLO.Q THEN
		fbAlLPHeaterTempLOLO.Clear(0, TRUE);
	END_IF
	IF trigFLPHPressHIHI.Q THEN
		fbAlLPHeaterPressHIHI.Clear(0, TRUE);
	END_IF
	IF trigFLPHPressHI.Q THEN
		fbAlLPHeaterPressHI.Clear(0, TRUE);
	END_IF
	IF trigFLPHPressLO.Q THEN
		fbAlLPHeaterPressLO.Clear(0, TRUE);
	END_IF
	IF trigFLPHPressLOLO.Q THEN
		fbAlLPHeaterPressLOLO.Clear(0, TRUE);
	END_IF
	IF trigFDeaerTempHIHI.Q THEN
		fbAlDeaeratorTempHIHI.Clear(0, TRUE);
	END_IF
	IF trigFDeaerTempHI.Q THEN
		fbAlDeaeratorTempHI.Clear(0, TRUE);
	END_IF
	IF trigFDeaerTempLO.Q THEN
		fbAlDeaeratorTempLO.Clear(0, TRUE);
	END_IF
	IF trigFDeaerTempLOLO.Q THEN
		fbAlDeaeratorTempLOLO.Clear(0, TRUE);
	END_IF
	IF trigFHPHTempHIHI.Q THEN
		fbAlHPHeaterTempHIHI.Clear(0, TRUE);
	END_IF
	IF trigFHPHTempHI.Q THEN
		fbAlHPHeaterTempHI.Clear(0, TRUE);
	END_IF
	IF trigFHPHTempLO.Q THEN
		fbAlHPHeaterTempLO.Clear(0, TRUE);
	END_IF
	IF trigFHPHTempLOLO.Q THEN
		fbAlHPHeaterTempLOLO.Clear(0, TRUE);
	END_IF
	IF trigFHPHPressHIHI.Q THEN
		fbAlHPHeaterPressHIHI.Clear(0, TRUE);
	END_IF
	IF trigFHPHPressHI.Q THEN
		fbAlHPHeaterPressHI.Clear(0, TRUE);
	END_IF
	IF trigFHPHPressLO.Q THEN
		fbAlHPHeaterPressLO.Clear(0, TRUE);
	END_IF
	IF trigFHPHPressLOLO.Q THEN
		fbAlHPHeaterPressLOLO.Clear(0, TRUE);
	END_IF
	IF trigFBoiTempHIHI.Q THEN
		fbAlBoilerTempHIHI.Clear(0, TRUE);
	END_IF
	IF trigFBoiTempHI.Q THEN
		fbAlBoilerTempHI.Clear(0, TRUE);
	END_IF
	IF trigFBoiTempLO.Q THEN
		fbAlBoilerTempLO.Clear(0, TRUE);
	END_IF
	IF trigFBoiTempLOLO.Q THEN
		fbAlBoilerTempLOLO.Clear(0, TRUE);
	END_IF
	IF trigFConTempHIHI.Q THEN
		fbAlCondenserTempHIHI.Clear(0, TRUE);
	END_IF
	IF trigFConTempHI.Q THEN
		fbAlCondenserTempHI.Clear(0, TRUE);
	END_IF
	IF trigFConTempLO.Q THEN
		fbAlCondenserTempLO.Clear(0, TRUE);
	END_IF
	IF trigFConTempLOLO.Q THEN
		fbAlCondenserTempLOLO.Clear(0, TRUE);
	END_IF
	IF trigFTurTempHIHI.Q THEN
		fbAlTurbineTempHIHI.Clear(0, TRUE);
	END_IF
	IF trigFTurTempHI.Q THEN
		fbAlTurbineTempHI.Clear(0, TRUE);
	END_IF
	IF trigFTurTempLO.Q THEN
		fbAlTurbineTempLO.Clear(0, TRUE);
	END_IF
	IF trigFTurTempLOLO.Q THEN
		fbAlTurbineTempLOLO.Clear(0, TRUE);
	END_IF
	IF trigFTurPressHIHI.Q THEN
		fbAlTurbinePressHIHI.Clear(0, TRUE);
	END_IF
	IF trigFTurPressHI.Q THEN
		fbAlTurbinePressHI.Clear(0, TRUE);
	END_IF
	IF trigFTurPressLO.Q THEN
		fbAlTurbinePressLO.Clear(0, TRUE);
	END_IF
	IF trigFTurPressLOLO.Q THEN
		fbAlTurbinePressLOLO.Clear(0, TRUE);
	END_IF
	IF trigFTurRotHIHI.Q THEN
		fbAlTurbineRotationHIHI.Clear(0, TRUE);
	END_IF
	IF trigFTurRotHI.Q THEN
		fbAlTurbineRotationHI.Clear(0, TRUE);
	END_IF
	IF trigFTurRotLO.Q THEN
		fbAlTurbineRotationLO.Clear(0, TRUE);
	END_IF
	IF trigFTurRotLOLO.Q THEN
		fbAlTurbineRotationLOLO.Clear(0, TRUE);
	END_IF
	
	IF bCfLPHeaterTempHIHI THEN
		bCfLPHeaterTempHIHI := FALSE;
		fbAlLPHeaterTempHIHI.Confirm(0);
	END_IF
	IF bCfLPHeaterTempHI THEN
		bCfLPHeaterTempHI := FALSE;
		fbAlLPHeaterTempHI.Confirm(0);
	END_IF
	IF bCfLPHeaterTempLO THEN
		bCfLPHeaterTempLO := FALSE;
		fbAlLPHeaterTempLO.Confirm(0);
	END_IF
	IF bCfLPHeaterTempLOLO THEN
		bCfLPHeaterTempLOLO := FALSE;
		fbAlLPHeaterTempLOLO.Confirm(0);
	END_IF
	IF bCfLPHeaterPressHIHI THEN
		bCfLPHeaterPressHIHI := FALSE;
		fbAlLPHeaterPressHIHI.Confirm(0);
	END_IF
	IF bCfLPHeaterPressHI THEN
		bCfLPHeaterPressHI := FALSE;
		fbAlLPHeaterPressHI.Confirm(0);
	END_IF
	IF bCfLPHeaterPressLO THEN
		bCfLPHeaterPressLO := FALSE;
		fbAlLPHeaterPressLO.Confirm(0);
	END_IF
	IF bCfLPHeaterPressLOLO THEN
		bCfLPHeaterPressLOLO := FALSE;
		fbAlLPHeaterPressLOLO.Confirm(0);
	END_IF
	IF bCfDeaeratorTempHIHI THEN
		bCfDeaeratorTempHIHI := FALSE;
		fbAlDeaeratorTempHIHI.Confirm(0);
	END_IF
	IF bCfDeaeratorTempHI THEN
		bCfDeaeratorTempHI := FALSE;
		fbAlDeaeratorTempHI.Confirm(0);
	END_IF
	IF bCfDeaeratorTempLO THEN
		bCfDeaeratorTempLO := FALSE;
		fbAlDeaeratorTempLO.Confirm(0);
	END_IF
	IF bCfDeaeratorTempLOLO THEN
		bCfDeaeratorTempLOLO := FALSE;
		fbAlDeaeratorTempLOLO.Confirm(0);
	END_IF
	IF bCfHPHeaterTempHIHI THEN
		bCfHPHeaterTempHIHI := FALSE;
		fbAlHPHeaterTempHIHI.Confirm(0);
	END_IF
	IF bCfHPHeaterTempHI THEN
		bCfHPHeaterTempHI := FALSE;
		fbAlHPHeaterTempHI.Confirm(0);
	END_IF
	IF bCfHPHeaterTempLO THEN
		bCfHPHeaterTempLO := FALSE;
		fbAlHPHeaterTempLO.Confirm(0);
	END_IF
	IF bCfHPHeaterTempLOLO THEN
		bCfHPHeaterTempLOLO := FALSE;
		fbAlHPHeaterTempLOLO.Confirm(0);
	END_IF
	IF bCfHPHeaterPressHIHI THEN
		bCfHPHeaterPressHIHI := FALSE;
		fbAlHPHeaterPressHIHI.Confirm(0);
	END_IF
	IF bCfHPHeaterPressHI THEN
		bCfHPHeaterPressHI := FALSE;
		fbAlHPHeaterPressHI.Confirm(0);
	END_IF
	IF bCfHPHeaterPressLO THEN
		bCfHPHeaterPressLO := FALSE;
		fbAlHPHeaterPressLO.Confirm(0);
	END_IF
	IF bCfHPHeaterPressLOLO THEN
		bCfHPHeaterPressLOLO := FALSE;
		fbAlHPHeaterPressLOLO.Confirm(0);
	END_IF
	IF bCfBoilerTempHIHI THEN
		bCfBoilerTempHIHI := FALSE;
		fbAlBoilerTempHIHI.Confirm(0);
	END_IF
	IF bCfBoilerTempHI THEN
		bCfBoilerTempHI := FALSE;
		fbAlBoilerTempHI.Confirm(0);
	END_IF
	IF bCfBoilerTempLO THEN
		bCfBoilerTempLO := FALSE;
		fbAlBoilerTempLO.Confirm(0);
	END_IF
	IF bCfBoilerTempLOLO THEN
		bCfBoilerTempLOLO := FALSE;
		fbAlBoilerTempLOLO.Confirm(0);
	END_IF
	IF bCfCondenserTempHIHI THEN
		bCfCondenserTempHIHI := FALSE;
		fbAlCondenserTempHIHI.Confirm(0);
	END_IF
	IF bCfCondenserTempHI THEN
		bCfCondenserTempHI := FALSE;
		fbAlCondenserTempHI.Confirm(0);
	END_IF
	IF bCfCondenserTempLO THEN
		bCfCondenserTempLO := FALSE;
		fbAlCondenserTempLO.Confirm(0);
	END_IF
	IF bCfCondenserTempLOLO THEN
		bCfCondenserTempLOLO := FALSE;
		fbAlCondenserTempLOLO.Confirm(0);
	END_IF
	IF bCfTurbineTempHIHI THEN
		bCfTurbineTempHIHI := FALSE;
		fbAlTurbineTempHIHI.Confirm(0);
	END_IF
	IF bCfTurbineTempHI THEN
		bCfTurbineTempHI := FALSE;
		fbAlTurbineTempHI.Confirm(0);
	END_IF
	IF bCfTurbineTempLO THEN
		bCfTurbineTempLO := FALSE;
		fbAlTurbineTempLO.Confirm(0);
	END_IF
	IF bCfTurbineTempLOLO THEN
		bCfTurbineTempLOLO := FALSE;
		fbAlTurbineTempLOLO.Confirm(0);
	END_IF
	IF bCfTurbinePressHIHI THEN
		bCfTurbinePressHIHI := FALSE;
		fbAlTurbinePressHIHI.Confirm(0);
	END_IF
	IF bCfTurbinePressHI THEN
		bCfTurbinePressHI := FALSE;
		fbAlTurbinePressHI.Confirm(0);
	END_IF
	IF bCfTurbinePressLO THEN
		bCfTurbinePressLO := FALSE;
		fbAlTurbinePressLO.Confirm(0);
	END_IF
	IF bCfTurbinePressLOLO THEN
		bCfTurbinePressLOLO := FALSE;
		fbAlTurbinePressLOLO.Confirm(0);
	END_IF
	IF bCfTurbineRotationHIHI THEN
		bCfTurbineRotationHIHI := FALSE;
		fbAlTurbineRotationHIHI.Confirm(0);
	END_IF
	IF bCfTurbineRotationHI THEN
		bCfTurbineRotationHI := FALSE;
		fbAlTurbineRotationHI.Confirm(0);
	END_IF
	IF bCfTurbineRotationLO THEN
		bCfTurbineRotationLO := FALSE;
		fbAlTurbineRotationLO.Confirm(0);
	END_IF
	IF bCfTurbineRotationLOLO THEN
		bCfTurbineRotationLOLO := FALSE;
		fbAlTurbineRotationLOLO.Confirm(0);
	END_IF

END_IF	
{endregion}

END_PROGRAM

// ---- POUs/UpdateInterface.TcPOU
PROGRAM UpdateInterface
VAR
	i: REAL := 0;
	fbton: TON;
END_VAR

Interfacex.ScadaInterface.Components.ForceFan1 := PnID.ForceFan1;
Interfacex.ScadaInterface.Components.ForceFan2 := PnID.ForceFan2;
Interfacex.ScadaInterface.Components.ForceFan3 := PnID.ForceFan3;

Interfacex.ScadaInterface.Components.CondensePump := PnID.CondensePump;
Interfacex.ScadaInterface.Components.SupplyPump := PnID.SupplyPump;
Interfacex.ScadaInterface.Components.CircularPump := PnID.CircularPump;
Interfacex.ScadaInterface.Components.InterPump := PnID.InterPump;

Interfacex.ScadaInterface.Components.LPHValve := PnID.LPHeaterValve;
Interfacex.ScadaInterface.Components.AirEjValve := PnID.AirEjectorValve;
Interfacex.ScadaInterface.Components.HPHValve := PnID.HPHeaterValve;
Interfacex.ScadaInterface.Components.TurbineValve := PnID.TurbineValve;

Interfacex.ScadaInterface.Components.Furnace.Temperature := Streams.InStream.Furnace_Temp;
Interfacex.ScadaInterface.Components.Furnace.InPercent := (Streams.InStream.ForceFan1_Speed/(3*Interfacex.Parameters.MaxSpeed_ForceFan1) + 
															Streams.InStream.ForceFan2_Speed/(3*Interfacex.Parameters.MaxSpeed_ForceFan2) +
															Streams.InStream.ForceFan3_Speed/(3*Interfacex.Parameters.MaxSpeed_ForceFan3))*100;
Interfacex.ScadaInterface.Components.LPHeater.Temperature := Streams.InStream.LPHeater_Temp;
Interfacex.ScadaInterface.Components.LPHeater.Pressure := Streams.InStream.LPHeater_Press;
Interfacex.ScadaInterface.Components.LPHeater.InPressure := Streams.InStream.CondensePump_Press;
Interfacex.ScadaInterface.Components.LPHeater.InFlow := Streams.InStream.CondensePump_Flow;
Interfacex.ScadaInterface.Components.Deaerator.Temperature := Streams.InStream.AirEjector_Temp;
Interfacex.ScadaInterface.Components.Deaerator.Pressure := Streams.InStream.AirEjector_Press;
Interfacex.ScadaInterface.Components.HPHeater.Temperature := Streams.InStream.HPHeater_Temp;
Interfacex.ScadaInterface.Components.HPHeater.Pressure := Streams.InStream.HPHeater_Press;
Interfacex.ScadaInterface.Components.HPHeater.InPressure := Streams.InStream.SupplyPump_Press;
Interfacex.ScadaInterface.Components.HPHeater.InFlow := Streams.InStream.SupplyPump_Flow;
Interfacex.ScadaInterface.Components.Boiler.Temperature := Streams.InStream.Boiler_Temp;
Interfacex.ScadaInterface.Components.Boiler.Pressure := Streams.InStream.Boiler_Press;
Interfacex.ScadaInterface.Components.Condenser.Temperature := Streams.InStream.Condenser_Temp;
Interfacex.ScadaInterface.Components.Condenser.InFlow := Streams.OutStream.CircularPump_OutFlow;//Streams.InStream.CircularPump_Flow;
Interfacex.ScadaInterface.Components.Turbine.Rotation := Streams.InStream.Turbine_Rotation;
Interfacex.ScadaInterface.Components.Turbine.HighTemperature := Streams.InStream.Turbine_HighTemp;
Interfacex.ScadaInterface.Components.Turbine.ImmediateTemperature := Streams.InStream.Turbine_ImmediateTemp;
Interfacex.ScadaInterface.Components.Turbine.OutTemperature := Streams.InStream.Turbine_OutTemp;
Interfacex.ScadaInterface.Components.Turbine.HighPressure := Streams.InStream.Turbine_HighPress;
Interfacex.ScadaInterface.Components.Turbine.ImmediatePressure := Streams.InStream.Turbine_ImmediatePress;
Interfacex.ScadaInterface.Components.Turbine.OutPressure := Streams.InStream.Turbine_OutPress;
Interfacex.ScadaInterface.Components.InterTank.HI := NOT PnID.bHI;
Interfacex.ScadaInterface.Components.InterTank.LO := PnID.bLO;
	
//Interfacex.ScadaInterface.Components.Furnace.Temperature := i * 1600;
//Interfacex.ScadaInterface.Components.Furnace.InPercent := i*100;
//Interfacex.ScadaInterface.Components.LPHeater.Temperature := i*160;
//Interfacex.ScadaInterface.Components.LPHeater.Pressure := i*36;
//Interfacex.ScadaInterface.Components.LPHeater.InPressure := i*50;
//Interfacex.ScadaInterface.Components.LPHeater.InFlow := i*36;
//Interfacex.ScadaInterface.Components.Deaerator.Temperature := i*250;
//Interfacex.ScadaInterface.Components.Deaerator.Pressure := i*36;
//Interfacex.ScadaInterface.Components.HPHeater.Temperature := i*320;
//Interfacex.ScadaInterface.Components.HPHeater.Pressure := i*320;
//Interfacex.ScadaInterface.Components.HPHeater.InPressure := i*36;
//Interfacex.ScadaInterface.Components.HPHeater.InFlow := i*50;
//Interfacex.ScadaInterface.Components.Boiler.Temperature := i*600;
//Interfacex.ScadaInterface.Components.Boiler.Pressure := i*260;
//Interfacex.ScadaInterface.Components.Condenser.Temperature := i*70;
//Interfacex.ScadaInterface.Components.Condenser.InFlow := i*100;
//Interfacex.ScadaInterface.Components.Turbine.Rotation := i*3600;
//Interfacex.ScadaInterface.Components.Turbine.HighTemperature := i*620;
//Interfacex.ScadaInterface.Components.Turbine.ImmediateTemperature := i*400;
//Interfacex.ScadaInterface.Components.Turbine.OutTemperature := i*180;
//Interfacex.ScadaInterface.Components.Turbine.HighPressure := i*60;
//Interfacex.ScadaInterface.Components.Turbine.ImmediatePressure := i*60;
//Interfacex.ScadaInterface.Components.Turbine.OutPressure := i*1;//Streams.InStream.Turbine_OutPress;

//fbton(IN:= NOT fbton.Q, PT:= T#100MS);
//IF (fbton.Q) THEN
//	i := i + 0.05;
//	IF i > 1 THEN
//		i := 0;
//	END_IF
//END_IF

END_PROGRAM

// ---- POUs/TanksSimulation.TcPOU
PROGRAM TanksSimulation
VAR_INPUT
	bStart AT %I* : BOOL;
	bEmerNC AT %I*: BOOL;
	bHI AT %I*: BOOL;
	bLO AT %I*: BOOL;
END_VAR	
VAR_OUTPUT
	bMotor1 AT %Q*: BOOL;
	bMotor2 AT %Q*: BOOL;
	bRun AT %Q*: BOOL;
	bErr AT %Q*: BOOL;
END_VAR
VAR
	bStateOn: BOOL := FALSE;
	bStateErr: BOOL := FALSE;
	trigStateOn: R_TRIG;
	bFirstScan: BOOL;
END_VAR

trigStateOn(CLK:= bStart);
IF trigStateOn.Q THEN
	IF bStateOn THEN
		bStateOn := FALSE;
	ELSE
		bStateOn := TRUE;
		bStateErr := FALSE;
		bMotor2 := TRUE;
	END_IF
END_IF

IF NOT bEmerNC THEN
	bStateErr := TRUE;
	bStateOn := FALSE;
END_IF

IF bStateOn THEN 
	IF NOT bHI THEN
		bMotor1:= FALSE;
		bMotor2:= TRUE;
	END_IF
	
	IF bLO THEN
		bMotor1:= TRUE;
		bMotor2:= FALSE;
	END_IF
ELSE
	bMotor1:= FALSE;
	bMotor2:= FALSE;
END_IF

bRun := bStateOn;
bErr := bStateErr;

END_PROGRAM
